FUNCTION_BLOCK "SINA_POS"   // FB1822, SCL
{ S7_Optimized_Access := 'TRUE' }
AUTHOR : DRVDPS7
FAMILY : DRIVES
NAME : SINA_POS
VERSION : 5.1
// stored: AutoNumber false, MemoryReserve 100, SetENOAutomatically false
   VAR_INPUT
      ModePos : Int := 0;   // 运行模式 1-相对；2-绝对；
      EnableAxis : Bool := 0;   // 使能驱动器
      CancelTraversing : Bool := 1;   // 0-取消当前任务运行;1-正常运行
      IntermediateStop : Bool := 1;   // 0-暂停当前的任务运行；1-正常运行
      Positive : Bool := 0;   // 正方向
      Negative : Bool := 0;   // 负方向
      Jog1 : Bool := 0;
      Jog2 : Bool := 0;
      FlyRef : Bool := 0;   // 激活被动寻零(CMMT不支持)
      AckError : Bool := 0;   // 故障复位
      ExecuteMode : Bool := 0;   // 激活ModPos模式
      Position : DInt := 0;   // 位置设定值或位置表行号
      Velocity : DInt := 0;   // 速度值
      OverV : Int := 100;   // 所有运动模式下的速度倍率（cmmt不支持）
      OverAcc : Int := 100;   // ModPos=1；2；3加速度百分比0-100
      OverDec : Int := 100;   // ModPos=1；2；3减速度百分比0-100
      ConfigEPos : DWord := 16#0000_0003;   // B0-3 功能位定义
      HWIDSTW : HW_IO := 0;   // CMMT 设备视图111报文硬件标识符
      HWIDZSW : HW_IO := 0;   // CMMT 设备视图111报文硬件标识符
   END_VAR
   VAR_OUTPUT
      AxisEnabled : Bool := 0;   // 驱动已经使能
      AxisPosOk : Bool := 0;   // 目标位置已到达
      AxisRef : Bool := 0;   // 已设置零点
      AxisWarn : Bool := 0;   // 驱动器报警
      AxisError : Bool := 0;   // 驱动器故障
      Lockout : Bool := 0;   // 驱动处于禁止接通状态，检查 ConfigEPos 第 0 位及第 1 位是否置 1
      ActVelocity : DInt := 0;   // 实际速度
      ActPosition : DInt := 0;   // 实际位置
      ActMode : Int := 0;   // 当前激活的模式
      EPosZSW1 : Word := 0;
      EPosZSW2 : Word := 0;
      ActWarn : Word := 0;   // 报警代码
      ActFault : Word := 0;   // 故障代码
      Error : Bool := 0;   // 功能块报错
      Status : Word := 0;   // 状态
      DiagID : Word := 0;   // 通信错误
   END_VAR
   VAR
      sbOff1Edge : Bool := 0;
      sbOff1 : Bool := 0;
      sbExecuteEdge : Bool := 0;
      sbExecute : Bool := 0;
      sbRefTypEdge : Bool := 0;
      sbRefTyp : Bool := 0;
      sbMdiStart : Bool := 0;
      sbMdiStartEdge : Bool := 0;
      sbRefStart : Bool := 0;
      sbJogInc : Bool := 0;
      sbReady : Bool := 0;
      sbIOp : Bool := 0;
      sbAccel : Bool := 0;
      sbDecel : Bool := 0;
      sbAlarm : Bool := 0;
      sbFault : Bool := 0;
      sbFWD : Bool := 0;
      sbBWD : Bool := 0;
      sbBusy : Bool := 0;
      swStatus : Word := 16#0000;
      swEPosZSW1 : Word := 16#0000;
      swEPosZSW2 : Word := 16#0000;
      siExecuteCyc : Int := 0;
      siRefTypCyc : Int := 0;
      siJogIncCyc : Int := 0;
      siMdiStartCyc : Int := 0;
      siRefActRetry : Int := 0;
      siModePos : Int := 0;
      siModePosMax : Int := 14;
      siCycWait : Int := 5;
      siRetryMax : Int := 15;
      sbModePos : Bool := 0;
      sxSendBuf : Struct
         STW1 : Word := WORD#16#0000;
         EPosSTW1 : Word := WORD#16#0000;
         EPosSTW2 : Word := WORD#16#0000;
         STW2 : Word := WORD#16#0000;
         OverrideV : Word := WORD#16#0000;
         Position : DWord := DWORD#16#0000_0000;
         Velocity : DWord := DWORD#16#0000_0000;
         OverrideA : Word := WORD#16#0000;
         OverrideD : Word := WORD#16#0000;
         Reserve : Word := WORD#16#0000;
      END_STRUCT;
      sxRecvBuf : Struct
         ZSW1 : Word := WORD#16#0000;
         EPosZSW1 : Word := WORD#16#0000;
         EPosZSW2 : Word := WORD#16#0000;
         ZSW2 : Word := WORD#16#0000;
         NotUsed : Word := WORD#16#0000;
         Position : DWord := DWORD#16#0000_0000;
         Velocity : DWord := DWORD#16#0000_0000;
         ErrNr : Word := WORD#16#0000;
         WarnNr : Word := WORD#16#0000;
         Reserve : Word := WORD#16#0000;
      END_STRUCT;
   END_VAR
   VAR_TEMP
      piRetSFC : Int;
      piCount : Int;
      swSendBuf : Array[0..11] of Word;
      swRecvBuf : Array[0..11] of Word;
   END_VAR
BEGIN

   //=============================================================================
   //SIEMENS AG
   //(c)Copyright 2017 All Rights Reserved
   //-----------------------------------------------------------------------------
   // Library: DriveLib
   // Tested with: S7-1516-3 PN/DP V1.8
   // Engineering: TIA Portal V14
   // Restrictions: -
   // Requirements: S7-1200 / S7-1500
   // Functionality: cyclic communication between a SINAMICS (Basic positioner)and a PLC
   //                If in HWConfig Std.TLG 111 is projected 12 PZD-words are exchanged
   //                in every bus cycle.
   //                The parametrisation of these words is described in the manual of the
   //                SINAMICS
   //=============================================================================

   // Betriebsart ermitteln
   IF #ModePos > #siModePosMax THEN

     #sbModePos := FALSE;
     #Error := True;
     #swStatus := 16#8202;//不正确的运行模式
   ELSIF #ModePos < 1 THEN

     #sbModePos := FALSE;
     #Error := True;
     #swStatus := 16#8202;//不正确的运行模式
   ELSE
     // Betriebsartenwechsel ist nur möglich, wenn die Achse nicht beschleunigt oder nicht verzögert 
     // und die Geschwindigkeit Null ist
     IF NOT #sbFWD AND NOT #sbBWD AND NOT #sbAccel AND NOT #sbDecel THEN

       #sbModePos := TRUE;
       #siModePos := #ModePos;

       // Fehler wieder zurücknehmen, wenn er mal ausgelöst wurde
       IF #swStatus = 16#8202 THEN
           #swStatus := 16#7002;//功能块正常执行
         #Error := False;
       END_IF;
     END_IF;
   END_IF;

   // Überprüfung der analogen Eingabewerte, ob sie innerhalb des möglichen Bereiches liegen
   // Geschwindigkeitsoverride (0% - 199%, 100% => W#16#4000)
   IF (#OverV < 0) OR (#OverV > 199) THEN
       #swStatus := 16#8203;//参数设置错误
     #Error := True;
   ELSE
     // Geschwindigkeitsoverride in den Sendepuffer eintragen
     #sxSendBuf.OverrideV := INT_TO_WORD(REAL_TO_INT(16384.0 * (INT_TO_REAL(#OverV) / 100.0)));
   END_IF;

   // Beschleunigungsoverride (0% - 100%, 100% => W#16#4000)
   IF (#OverAcc < 0) OR (#OverAcc > 100) THEN
       #swStatus := 16#8203;//参数设置错误
     #Error := True;
   ELSE
     // Beschleunigungsoverride in den Sendepuffer eintragen
     #sxSendBuf.OverrideA := INT_TO_WORD(REAL_TO_INT(16384.0 * (INT_TO_REAL(#OverAcc) / 100.0)));
   END_IF;

   // Verzögerungsoverride (0% - 100%, 100% => W#16#4000)
   IF (#OverDec < 0) OR (#OverDec > 100) THEN
       #swStatus := 16#8203;//参数设置错误
     #Error := True;
   ELSE
     // Verzögerungsoverride in den Sendepuffer eintragen
     #sxSendBuf.OverrideD := INT_TO_WORD(REAL_TO_INT(16384.0 * (INT_TO_REAL(#OverDec) / 100.0)));
   END_IF;

   // Fehler wieder zurücknehmen, wenn er mal ausgelöst wurde
   IF NOT (#OverV < 0) AND NOT (#OverV > 199) AND NOT (#OverAcc < 0) AND NOT (#OverAcc > 100) AND
     NOT (#OverDec < 0) AND NOT (#OverDec > 100) THEN
     IF #swStatus = 16#8203 THEN
       #swStatus := 16#7002;
       #Error := False;
     END_IF;
   END_IF;

   // Positionssollwert
   // Positionssollwert in den Sendepuffer eintragen
   #sxSendBuf.Position := DINT_TO_DWORD(#Position);

   // Geschwindigkeitssollwert (Begrenzung / Überwachung
   // Geschwindigkeitssollwert in den Sendepuffer eintragen
   #sxSendBuf.Velocity := DINT_TO_DWORD(#Velocity);

   // Einschalten bzw. Ausschalten des Antriebes erkennen
   IF #EnableAxis AND NOT #sbOff1Edge AND NOT #sbBusy AND #sbModePos THEN
     #sbOff1 := True;
   END_IF;
   // Einschalten bzw. Ausschalten des Antriebes Flanke merken
   #sbOff1Edge := #EnableAxis AND NOT #sbBusy;

   // Einschaltflankenmerker wieder zurücksetzen
   IF NOT #EnableAxis THEN
     #sbOff1 := False;
   END_IF;

   // Fliegendes Referenzieren aktivieren erkennen
   IF #FlyRef AND NOT #sbRefTypEdge THEN
     #sbRefTyp := True;
   END_IF;
   // Fliegendes Referenzieren aktivieren Flanke merken
   #sbRefTypEdge := #FlyRef;

   // Fliegendes Referenzieren Flankenmerker wieder zurücksetzen
   IF NOT #FlyRef THEN
     #sbRefTyp := False;
     #siRefTypCyc := 0;
   END_IF;

   // Verfahrauftrag aktivieren erkennen
   IF #ExecuteMode AND NOT #sbExecuteEdge THEN
     #sbExecute := True;
   END_IF;
   // Verfahrauftrag aktivieren Flanke merken
   #sbExecuteEdge := #ExecuteMode;

   // Verfahrauftragflankenmerker wieder zurücksetzen
   IF NOT #ExecuteMode THEN
     #sbExecute := False;
     #siExecuteCyc := 0;
   END_IF;

   // Betriebsart MDI / Sollwertdirektvorgabe Flanke merken
   (*IF #sxSendBuf.sxEPosSTW1.MdiStart AND NOT #sbMdiStartEdge THEN
             #sbMdiStart := True;
         END_IF;
         // Betriebsart MDI / Sollwertdirektvorgabe Flanke merken
         #sbMdiStartEdge := #sxSendBuf.sxEPosSTW1.MdiStart AND NOT #Busy;*)

   // Verfahrauftragflankenmerker wieder zurücksetzen
   (*IF NOT #sxSendBuf.sxEPosSTW1.MdiStart THEN
             #sbMdiStart := False;
             #siMdiStartCyc := 0;
         END_IF;*)

   IF #sxSendBuf.EPosSTW1.%X15 AND NOT #sbMdiStartEdge THEN
     #sbMdiStart := True;
   END_IF;
   // Betriebsart MDI / Sollwertdirektvorgabe Flanke merken
   #sbMdiStartEdge := #sxSendBuf.EPosSTW1.%X15 AND NOT #sbBusy;

   // Verfahrauftragflankenmerker wieder zurücksetzen
   IF NOT #sxSendBuf.EPosSTW1.%X15 THEN
     #sbMdiStart := False;
     #siMdiStartCyc := 0;
   END_IF;

   // Schreibdaten zusammenstellen
   // Steuerword STW1 für alle Betriebsart aufbereiten
   (*#sxSendBuf.sxSTW1.RejTrvTsk        := #RejTrvTsk;
         #sxSendBuf.sxSTW1.IntMStop         := #IntMStop;
         #sxSendBuf.sxSTW1.AckFault         := #AckFlt;*)

   #sxSendBuf.STW1.%X4 := #CancelTraversing;
   #sxSendBuf.STW1.%X5 := #IntermediateStop;
   #sxSendBuf.STW1.%X7 := #AckError;
   #sxSendBuf.STW1.%X1 := TRUE;
   #sxSendBuf.STW1.%X2 := TRUE;
   #sxSendBuf.STW1.%X3 := TRUE;
   #sxSendBuf.STW1.%X10 := TRUE;

   // Hauptbetriebsart "Positionieren / manueller Sollwertvorgabe (MDI)" 
   // Betriebsart "Positionieren Relativ positiv" oder "Positionieren Relativ negativ"
   IF (#siModePos = 1 AND #sbModePos) THEN

     // Antrieb einschalten
     //#sxSendBuf.sxSTW1.Off1 := #sbOff1;
     #sxSendBuf.STW1.%X0 := #sbOff1;

     // nicht verwendete Signale für den 1. Schritt und eventuell weitere Schritte
     (*#sxSendBuf.sxSTW1.Jog1          := False;
             #sxSendBuf.sxSTW1.Jog2          := False;
             #sxSendBuf.sxEPosSTW1.MdiTyp    := False;
             #sxSendBuf.sxEPosSTW1.MdiPos    := False;
             #sxSendBuf.sxEPosSTW1.MdiNeg    := False;
             #sxSendBuf.sxEPosSTW1.MdiSetup  := False;
             #sxSendBuf.sxEPosSTW2.SetRefPt  := False;
             #sxSendBuf.sxEPosSTW2.JogInc    := False;
             #sxSendBuf.sxEPosSTW2.RefStDi   := False;
             #sxSendBuf.sxSTW1.RefStart      := False;
             #sxSendBuf.sxEPosSTW2.RefTyp    := False;
             #sxSendBuf.sxEPosSTW1.MdiStart  := False;*)
     #sxSendBuf.STW1.%X8 := False;
     #sxSendBuf.STW1.%X9 := False;
     #sxSendBuf.EPosSTW1.%X8 := False;
     #sxSendBuf.EPosSTW1.%X9 := False;
     #sxSendBuf.EPosSTW1.%X10 := False;
     #sxSendBuf.EPosSTW1.%X14 := False;
     #sxSendBuf.EPosSTW2.%X1 := False;
     #sxSendBuf.EPosSTW2.%X5 := False;
     #sxSendBuf.EPosSTW2.%X9 := False;
     #sxSendBuf.STW1.%X11 := False;
     #sxSendBuf.EPosSTW2.%X8 := False;
     #sxSendBuf.EPosSTW1.%X15 := False;


     // Nach dem Einschalten des Antriebes, prüfen ob der Antrieb betriebsbereit, in Operation ohne Fehler und Warnung ist, 
     // dann die Betriebsart MDI / Sollwertvorgabe Start gesetzt werden
     IF #sbOff1 AND #sbReady AND #sbIOp AND NOT #sbFault THEN

       // Betriebsart MDI / Sollwertdirektvorgabe setzen
       //#sxSendBuf.sxEPosSTW1.MdiStart := True;
       #sxSendBuf.EPosSTW1.%X15 := True;

       // Positioniertyp auf relatives Positionieren stellen 
       //#sxSendBuf.sxEPosSTW1.MdiTyp := False;
       #sxSendBuf.EPosSTW1.%X8 := False;

       // die Richtungswahl für das Positionieren auf positive Richtung oder negative Richtung einstellen
       IF #Positive AND NOT #Negative THEN

         // positive Richtung
         //#sxSendBuf.sxEPosSTW1.MdiPos := True;
         #sxSendBuf.EPosSTW1.%X9 := True;

         // negative Richtung
         //#sxSendBuf.sxEPosSTW1.MdiNeg := False;
         #sxSendBuf.EPosSTW1.%X10 := False;

         // die Richtungswahl für das Positionieren auf negative Richtung einstellen                
       ELSIF NOT #Positive AND #Negative THEN

         // positive Richtung
         //#sxSendBuf.sxEPosSTW1.MdiPos := False;
         #sxSendBuf.EPosSTW1.%X9 := False;

         // negative Richtung
         //#sxSendBuf.sxEPosSTW1.MdiNeg := True;
         #sxSendBuf.EPosSTW1.%X10 := True;

         // die Richtungswahl für das Positionieren auf keine Richtung einstellen                
       ELSE

         // positive Richtung
         //#sxSendBuf.sxEPosSTW1.MdiPos := False;
         #sxSendBuf.EPosSTW1.%X9 := False;

         // negative Richtung
         //#sxSendBuf.sxEPosSTW1.MdiNeg := False;
         #sxSendBuf.EPosSTW1.%X10 := False;

       END_IF;

       // Nach dem Einschalten des Antriebes und dem Betriebsart MDI / Sollwertvorgabe starten, 
       // ein Paar Zyklen warten bevor die Flanke für die Sollwertübernahme MDI gesetzt werden kann
       IF #sbMdiStart AND (#siMdiStartCyc < #siCycWait) THEN
         #siMdiStartCyc := #siMdiStartCyc + 1;
       ELSE
         // Flanke Sollwertübernahme MDI
         //#sxSendBuf.sxSTW1.TrvStart := #Execute;
         #sxSendBuf.STW1.%X6 := #ExecuteMode;

       END_IF;

       // "Fliegendes Referentieren" aktivieren
       // "Fliegendes Referenzieren" erst nach Einschalten des Antriebes möglich
       IF #sbRefTyp THEN

         // Referenziertyp auf "Fliegendes Referenzieren" einstellen
         //#sxSendBuf.sxEPosSTW2.RefTyp := True;
         #sxSendBuf.EPosSTW2.%X8 := True;

         // Nach der Anwahl des Referenziertyps "Fliegendes Referenzieren", 
         // ein Zyklus später kann das Referenzieren gestartet
         IF (#siRefTypCyc = 0) THEN
           #siRefTypCyc := #siRefTypCyc + 1;
         ELSE
           // Referenzieren starten
           //#sxSendBuf.sxSTW1.RefStart := True;
           #sxSendBuf.STW1.%X11 := True;

         END_IF;
       END_IF;
     END_IF;

     // Betriebsart "Positionieren Absolut" oder "Positonieren Absolut positiv" oder "Positionieren Absolut negativ"
   ELSIF #siModePos = 2 AND #sbModePos THEN

     // Antrieb einschalten
     //#sxSendBuf.sxSTW1.Off1 := #sbOff1;
     #sxSendBuf.STW1.%X0 := #sbOff1;

     // nicht verwendete Signale für den 1. Schritt und eventuell weitere Schritte
     (*#sxSendBuf.sxSTW1.Jog1         := False;
             #sxSendBuf.sxSTW1.Jog2         := False;
             #sxSendBuf.sxEPosSTW1.MdiTyp   := False;
             #sxSendBuf.sxEPosSTW1.MdiPos   := False;
             #sxSendBuf.sxEPosSTW1.MdiNeg   := False;
             #sxSendBuf.sxEPosSTW1.MdiSetup := False;
             #sxSendBuf.sxEPosSTW2.SetRefPt := False;
             #sxSendBuf.sxEPosSTW2.JogInc   := False;
             #sxSendBuf.sxEPosSTW2.RefStDi  := False;
             #sxSendBuf.sxSTW1.RefStart     := False;
             #sxSendBuf.sxEPosSTW2.RefTyp   := False;
             #sxSendBuf.sxEPosSTW1.MdiStart := False;*)
     #sxSendBuf.STW1.%X8 := False;
     #sxSendBuf.STW1.%X9 := False;
     #sxSendBuf.EPosSTW1.%X8 := False;
     #sxSendBuf.EPosSTW1.%X9 := False;
     #sxSendBuf.EPosSTW1.%X10 := False;
     #sxSendBuf.EPosSTW1.%X14 := False;
     #sxSendBuf.EPosSTW2.%X1 := False;
     #sxSendBuf.EPosSTW2.%X5 := False;
     #sxSendBuf.EPosSTW2.%X9 := False;
     #sxSendBuf.STW1.%X11 := False;
     #sxSendBuf.EPosSTW2.%X8 := False;
     #sxSendBuf.EPosSTW1.%X15 := False;

     // Nach dem Einschalten des Antriebes, prüfen ob der Antrieb betriebsbereit, in Operation ohne Fehler und Warnung ist, 
     // dann die Betriebsart MDI / Sollwertvorgabe Start gesetzt werden
     IF #sbOff1 AND #sbReady AND #sbIOp AND NOT #sbFault THEN

       // Betriebsart MDI / Sollwertdirektvorgabe setzen
       //#sxSendBuf.sxEPosSTW1.MdiStart := True;
       #sxSendBuf.EPosSTW1.%X15 := True;

       // Positioniertyp auf absolutes Positionieren stellen 
       //#sxSendBuf.sxEPosSTW1.MdiTyp := True;
       #sxSendBuf.EPosSTW1.%X8 := True;

       // die Richtungswahl für das Positionieren auf positive Richtung oder negative Richtung einstellen
       IF #Positive AND NOT #Negative THEN

         // positive Richtung
         //#sxSendBuf.sxEPosSTW1.MdiPos := True;
         #sxSendBuf.EPosSTW1.%X9 := True;

         // negative Richtung
         //#sxSendBuf.sxEPosSTW1.MdiNeg := False;
         #sxSendBuf.EPosSTW1.%X10 := False;

         // die Richtungswahl für das Positionieren auf negative Richtung einstellen                
       ELSIF NOT #Positive AND #Negative THEN

         // positive Richtung
         //#sxSendBuf.sxEPosSTW1.MdiPos := False;
         #sxSendBuf.EPosSTW1.%X9 := False;

         // negative Richtung
         //#sxSendBuf.sxEPosSTW1.MdiNeg := True;
         #sxSendBuf.EPosSTW1.%X10 := True;

         // die Richtungswahl für das Positionieren auf keine Richtung einstellen                
       ELSE

         // positive Richtung
         //#sxSendBuf.sxEPosSTW1.MdiPos := False;
         #sxSendBuf.EPosSTW1.%X9 := False;

         // negative Richtung
         //#sxSendBuf.sxEPosSTW1.MdiNeg := False;
         #sxSendBuf.EPosSTW1.%X10 := False;

       END_IF;

       // Nach dem Einschalten des Antriebes und dem Betriebsart MDI / Sollwertvorgabe starten, 
       // ein Paar Zyklen warten bevor die Flanke für die Sollwertübernahme MDI gesetzt werden kann
       IF #sbMdiStart AND (#siMdiStartCyc < #siCycWait) THEN
         #siMdiStartCyc := #siMdiStartCyc + 1;
       ELSE
         // Flanke Sollwertübernahme MDI
         //#sxSendBuf.sxSTW1.TrvStart := #Execute;
         #sxSendBuf.STW1.%X6 := #ExecuteMode;

       END_IF;

       // "Fliegendes Referentieren" aktivieren
       // "Fliegendes Referenzieren" erst nach Einschalten des Antriebes möglich
       IF #sbRefTyp THEN

         // Referenziertyp auf "Fliegendes Referenzieren" einstellen
         //#sxSendBuf.sxEPosSTW2.RefTyp := True;
         #sxSendBuf.EPosSTW2.%X8 := True;

         // Nach der Anwahl des Referenziertyps "Fliegendes Referenzieren", 
         // ein Zyklus später kann das Referenzieren gestartet
         IF (#siRefTypCyc = 0) THEN
           #siRefTypCyc := #siRefTypCyc + 1;
         ELSE
           // Referenzieren starten
           //#sxSendBuf.sxSTW1.RefStart := True;
           #sxSendBuf.STW1.%X11 := True;

         END_IF;
       END_IF;
     END_IF;

     // Betriebsart "Positionieren als Einrichten positiv" oder "Positionieren als Einrichten negativ"
   ELSIF #siModePos = 3 AND #sbModePos THEN

     // Antrieb einschalten
     //#sxSendBuf.sxSTW1.Off1 := #sbOff1;
     #sxSendBuf.STW1.%X0 := #sbOff1;

     // nicht verwendete Signale für den 1. Schritt und eventuell weitere Schritte
     (*#sxSendBuf.sxSTW1.Jog1           := False;
             #sxSendBuf.sxSTW1.Jog2           := False;
             #sxSendBuf.sxEPosSTW1.MdiTyp     := False;
             #sxSendBuf.sxEPosSTW1.MdiPos     := False;
             #sxSendBuf.sxEPosSTW1.MdiNeg     := False;
             #sxSendBuf.sxEPosSTW1.MdiSetup   := False;
             #sxSendBuf.sxEPosSTW2.SetRefPt   := False;
             #sxSendBuf.sxEPosSTW2.JogInc     := False;
             #sxSendBuf.sxEPosSTW2.RefStDi    := False;
             #sxSendBuf.sxSTW1.RefStart       := False;
             #sxSendBuf.sxEPosSTW2.RefTyp     := False;
             #sxSendBuf.sxEPosSTW1.MdiStart   := False;*)
     #sxSendBuf.STW1.%X8 := False;
     #sxSendBuf.STW1.%X9 := False;
     #sxSendBuf.EPosSTW1.%X8 := False;
     #sxSendBuf.EPosSTW1.%X9 := False;
     #sxSendBuf.EPosSTW1.%X10 := False;
     #sxSendBuf.EPosSTW1.%X14 := False;
     #sxSendBuf.EPosSTW2.%X1 := False;
     #sxSendBuf.EPosSTW2.%X5 := False;
     #sxSendBuf.EPosSTW2.%X9 := False;
     #sxSendBuf.STW1.%X11 := False;
     #sxSendBuf.EPosSTW2.%X8 := False;
     #sxSendBuf.EPosSTW1.%X15 := False;

     // Nach dem Einschalten des Antriebes, prüfen ob der Antrieb betriebsbereit, in Operation ohne Fehler und Warnung ist, 
     // dann die Betriebsart MDI / Sollwertvorgabe Start gesetzt werden
     IF #sbOff1 AND #sbReady AND #sbIOp AND NOT #sbFault THEN

       // Betriebsart MDI / Sollwertdirektvorgabe setzen
       //#sxSendBuf.sxEPosSTW1.MdiStart := True;
       #sxSendBuf.EPosSTW1.%X15 := True;

       // Positioniertyp auf absolutes Positionieren stellen 
       //#sxSendBuf.sxEPosSTW1.MdiTyp := True;
       #sxSendBuf.EPosSTW1.%X8 := True;

       // die Anwahl für MDI Modus auf Einrichten einstellen
       //#sxSendBuf.sxEPosSTW1.MdiSetup := True;
       #sxSendBuf.EPosSTW1.%X14 := True;

       // die Richtungswahl für das Positionieren auf positive Richtung oder negative Richtung einstellen
       IF #Positive AND NOT #Negative THEN

         // positive Richtung
         //#sxSendBuf.sxEPosSTW1.MdiPos := True;
         #sxSendBuf.EPosSTW1.%X9 := True;

         // negative Richtung
         //#sxSendBuf.sxEPosSTW1.MdiNeg := False;
         #sxSendBuf.EPosSTW1.%X10 := False;

         // die Richtungswahl für das Positionieren auf negative Richtung einstellen                
       ELSIF NOT #Positive AND #Negative THEN

         // positive Richtung
         //#sxSendBuf.sxEPosSTW1.MdiPos := False;
         #sxSendBuf.EPosSTW1.%X9 := False;

         // negative Richtung
         //#sxSendBuf.sxEPosSTW1.MdiNeg := True;
         #sxSendBuf.EPosSTW1.%X10 := True;

         // die Richtungswahl für das Positionieren auf keine Richtung einstellen                
       ELSE

         // positive Richtung
         //#sxSendBuf.sxEPosSTW1.MdiPos := False;
         #sxSendBuf.EPosSTW1.%X9 := False;

         // negative Richtung
         //#sxSendBuf.sxEPosSTW1.MdiNeg := False;
         #sxSendBuf.EPosSTW1.%X10 := False;

       END_IF;

       // Nach dem Einschalten des Antriebes und dem Betriebsart MDI / Sollwertvorgabe starten, 
       // ein Paar Zyklen warten bevor die Flanke für die Sollwertübernahme MDI gesetzt werden kann
       IF #sbMdiStart AND (#siMdiStartCyc < #siCycWait) THEN
         #siMdiStartCyc := #siMdiStartCyc + 1;
       ELSE
         // Flanke Sollwertübernahme MDI
         //#sxSendBuf.sxSTW1.TrvStart := #Execute;
         #sxSendBuf.STW1.%X6 := #ExecuteMode;

       END_IF;

       // "Fliegendes Referentieren" aktivieren
       // "Fliegendes Referenzieren" erst nach Einschalten des Antriebes möglich
       IF #sbRefTyp THEN

         // Referenziertyp auf "Fliegendes Referenzieren" einstellen
         //#sxSendBuf.sxEPosSTW2.RefTyp := True;
         #sxSendBuf.EPosSTW2.%X8 := True;

         // Nach der Anwahl des Referenziertyps "Fliegendes Referenzieren", 
         // ein Zyklus später kann das Referenzieren gestartet
         IF (#siRefTypCyc = 0) THEN
           #siRefTypCyc := #siRefTypCyc + 1;
         ELSE
           // Referenzieren starten
           //#sxSendBuf.sxSTW1.RefStart := True;
           #sxSendBuf.STW1.%X11 := True;

         END_IF;
       END_IF;
     END_IF;

     // Hauptbetriebsart "Referenzieren" (Reference)
     // Betriebsart "Referenzieren - Referenzpunktfahrt positiv" oder "Referenzieren - Referenzpunktfahrt negativ"
   ELSIF #siModePos = 4 AND #sbModePos THEN

     // Antrieb einschalten
     //#sxSendBuf.sxSTW1.Off1 := #sbOff1;
     #sxSendBuf.STW1.%X0 := #sbOff1;

     // nicht verwendete Signale für den 1. Schritt und eventuell weitere Schritte
     (*#sxSendBuf.sxSTW1.Jog1         := False;
             #sxSendBuf.sxSTW1.Jog2         := False;
             #sxSendBuf.sxEPosSTW1.MdiStart := False;
             #sxSendBuf.sxEPosSTW2.SetRefPt := False;
             #sxSendBuf.sxEPosSTW2.JogInc   := False;
             #sxSendBuf.sxEPosSTW2.RefTyp   := False;
             #sxSendBuf.sxSTW1.RefStart     := False;
             #sxSendBuf.sxEPosSTW2.RefStDi  := False;*)
     #sxSendBuf.STW1.%X8 := False;
     #sxSendBuf.STW1.%X9 := False;
     #sxSendBuf.EPosSTW1.%X15 := False;
     #sxSendBuf.EPosSTW2.%X1 := False;
     #sxSendBuf.EPosSTW2.%X5 := False;
     #sxSendBuf.EPosSTW2.%X8 := False;
     #sxSendBuf.STW1.%X11 := False;
     #sxSendBuf.EPosSTW2.%X9 := False;

     // Nach dem Einschalten des Antriebes, prüfen ob der Antrieb betriebsbereit, in Operation ohne Fehler und Warnung ist, 
     // dann die Betriebsart MDI / Sollwertvorgabe Start gesetzt werden
     IF #sbOff1 AND #sbReady AND #sbIOp AND NOT #sbFault THEN

       // Referenzieren starten
       //#sxSendBuf.sxSTW1.RefStart := #Execute;
       #sxSendBuf.STW1.%X11 := #ExecuteMode;

       // die Richtungswahl für das Referenzpunktfahrt positiv einstellen
       IF #Positive AND NOT #Negative THEN

         // positive Referenzpunktfahrt
         //#sxSendBuf.sxEPosSTW2.RefStDi := False;
         #sxSendBuf.EPosSTW2.%X9 := False;

         // die Richtungswahl für das Referenzpunktfahrt negativ einstellen                
       ELSIF NOT #Positive AND #Negative THEN

         // negative Referenzpunktfahrt
         //#sxSendBuf.sxEPosSTW2.RefStDi := True;
         #sxSendBuf.EPosSTW2.%X9 := True;

       END_IF;
     END_IF;

     // Betriebsart "Referenzieren - Referenzpunkt setzen"
   ELSIF #siModePos = 5 AND #sbModePos THEN

     // Antrieb einschalten
     //#sxSendBuf.sxSTW1.Off1 := #sbOff1;
     #sxSendBuf.STW1.%X0 := #sbOff1;

     // nicht verwendete Signale für den 1. Schritt und eventuell weitere Schritte
     (*#sxSendBuf.sxSTW1.Jog1          := False;
             #sxSendBuf.sxSTW1.Jog2          := False;
             #sxSendBuf.sxSTW1.RefStart      := False;
             #sxSendBuf.sxEPosSTW1.MdiStart  := False;
             #sxSendBuf.sxEPosSTW2.JogInc    := False;
             #sxSendBuf.sxEPosSTW2.RefTyp    := False;
             #sxSendBuf.sxEPosSTW2.RefStDi   := False;
             #sxSendBuf.sxEPosSTW2.SetRefPt  := False;*)
     #sxSendBuf.STW1.%X8 := False;
     #sxSendBuf.STW1.%X9 := False;
     #sxSendBuf.STW1.%X11 := False;
     #sxSendBuf.EPosSTW1.%X15 := False;
     #sxSendBuf.EPosSTW2.%X5 := False;
     #sxSendBuf.EPosSTW2.%X8 := False;
     #sxSendBuf.EPosSTW2.%X9 := False;
     #sxSendBuf.EPosSTW2.%X1 := False;

     // Nach dem Einschalten des Antriebes, prüfen ob der Antrieb betriebsbereit, in Operation ohne Fehler und Warnung ist, 
     // dann die Betriebsart MDI / Sollwertvorgabe Start gesetzt werden
     IF NOT #sbFault THEN

       // Referenzpunktfahrt negativ
       //#sxSendBuf.sxEPosSTW2.SetRefPt := #Execute;
       #sxSendBuf.EPosSTW2.%X1 := #ExecuteMode;

     END_IF;

     // Hauptbetriebsart "Verfahrsätze" (Traversing Blocks)
   ELSIF #siModePos = 6 AND #sbModePos THEN

     // Antrieb einschalten
     //#sxSendBuf.sxSTW1.Off1 := #sbOff1;
     #sxSendBuf.STW1.%X0 := #sbOff1;

     // nicht verwendete Signale für den 1. Schritt und eventuell weitere Schritte
     (*#sxSendBuf.sxSTW1.Jog1          := False;
             #sxSendBuf.sxSTW1.Jog2          := False;
             #sxSendBuf.sxEPosSTW1.MdiTyp    := False;
             #sxSendBuf.sxEPosSTW1.MdiPos    := False;
             #sxSendBuf.sxEPosSTW1.MdiNeg    := False;
             #sxSendBuf.sxEPosSTW1.MdiSetup  := False;
             #sxSendBuf.sxEPosSTW2.SetRefPt  := False;
             #sxSendBuf.sxEPosSTW2.JogInc    := False;
             #sxSendBuf.sxEPosSTW2.RefStDi   := False;
             #sxSendBuf.sxEPosSTW2.RefTyp    := False;
             #sxSendBuf.sxSTW1.RefStart      := False;
             #sxSendBuf.sxEPosSTW1.TrvBit0   := False;
             #sxSendBuf.sxEPosSTW1.TrvBit1   := False;
             #sxSendBuf.sxEPosSTW1.TrvBit2   := False;
             #sxSendBuf.sxEPosSTW1.TrvBit3   := False;
             #sxSendBuf.sxEPosSTW1.TrvBit4   := False;
             #sxSendBuf.sxEPosSTW1.TrvBit5   := False;
             #sxSendBuf.sxEPosSTW1.MdiStart  := False;*)
     #sxSendBuf.STW1.%X8 := False;
     #sxSendBuf.STW1.%X9 := False;
     #sxSendBuf.EPosSTW1.%X8 := False;
     #sxSendBuf.EPosSTW1.%X9 := False;
     #sxSendBuf.EPosSTW1.%X10 := False;
     #sxSendBuf.EPosSTW1.%X14 := False;
     #sxSendBuf.EPosSTW2.%X1 := False;
     #sxSendBuf.EPosSTW2.%X5 := False;
     #sxSendBuf.EPosSTW2.%X9 := False;
     #sxSendBuf.EPosSTW2.%X8 := False;
     #sxSendBuf.STW1.%X11 := False;
     #sxSendBuf.EPosSTW1.%X0 := False;
     #sxSendBuf.EPosSTW1.%X1 := False;
     #sxSendBuf.EPosSTW1.%X2 := False;
     #sxSendBuf.EPosSTW1.%X3 := False;
     #sxSendBuf.EPosSTW1.%X4 := False;
     #sxSendBuf.EPosSTW1.%X5 := False;
     #sxSendBuf.EPosSTW1.%X15 := False;

     // Bei der Auswahl der Verfahrsätze entspricht die Position der Verfahrensatznummer 
     // Verfahrsatznummer aus der Position ermitteln und in die einzelnen Bit's aufteilen
     // Es sind die Verfahrsatznummern 0 - 63 möglich
     IF (DINT_TO_INT(#Position) < 0) OR (DINT_TO_INT(#Position) > 63) THEN
       // Fehler, ungültiger Verfahrsatznummer
       #swStatus := 16#8204;
       #Error := True;
     ELSE
       // Fehler wieder zurücknehmen, wenn er mal ausgelöst wurde
       IF #swStatus = 16#8204 THEN
         #swStatus := 16#7002;
         #Error := False;
       END_IF;

       // Verfahrsatznummer Bit 0 ermitteln
       IF (DINT_TO_WORD(#Position) AND W#16#01) = W#16#01 THEN
         //#sxSendBuf.sxEPosSTW1.TrvBit0 := True;
         #sxSendBuf.EPosSTW1.%X0 := True;
       END_IF;

       // Verfahrsatznummer Bit 1 ermitteln
       IF (DINT_TO_WORD(#Position) AND W#16#02) = W#16#02 THEN
         //#sxSendBuf.sxEPosSTW1.TrvBit1 := True;
         #sxSendBuf.EPosSTW1.%X1 := True;
       END_IF;

       // Verfahrsatznummer Bit 2 ermitteln
       IF (DINT_TO_WORD(#Position) AND W#16#04) = W#16#04 THEN
         //#sxSendBuf.sxEPosSTW1.TrvBit2 := True;
         #sxSendBuf.EPosSTW1.%X2 := True;
       END_IF;

       // Verfahrsatznummer Bit 3 ermitteln
       IF (DINT_TO_WORD(#Position) AND W#16#08) = W#16#08 THEN
         //#sxSendBuf.sxEPosSTW1.TrvBit3 := True;
         #sxSendBuf.EPosSTW1.%X3 := True;
       END_IF;

       // Verfahrsatznummer Bit 4 ermitteln
       IF (DINT_TO_WORD(#Position) AND W#16#10) = W#16#10 THEN
         //#sxSendBuf.sxEPosSTW1.TrvBit4 := True;
         #sxSendBuf.EPosSTW1.%X4 := True;
       END_IF;

       // Verfahrsatznummer Bit 5 ermitteln
       IF (DINT_TO_WORD(#Position) AND W#16#20) = W#16#20 THEN
         //#sxSendBuf.sxEPosSTW1.TrvBit5 := True;
         #sxSendBuf.EPosSTW1.%X5 := True;
       END_IF;

       // Nach dem Einschalten des Antriebes, prüfen ob der Antrieb betriebsbereit, in Operation ohne Fehler und Warnung ist, 
       // dann die Betriebsart MDI / Sollwertvorgabe Start gesetzt werden
       IF #sbOff1 AND #sbReady AND #sbIOp AND NOT #sbFault THEN

         // Positioniertyp auf absolutes Positionieren stellen 
         //#sxSendBuf.sxEPosSTW1.MdiTyp := True;
         #sxSendBuf.EPosSTW1.%X8 := True;

         // die Richtungswahl für das Positionieren auf positive Richtung einstellen
         //#sxSendBuf.sxEPosSTW1.MdiPos := True;
         #sxSendBuf.EPosSTW1.%X9 := True;

         // die Richtungswahl für das Positionieren auf negative Richtung abstellen
         //#sxSendBuf.sxEPosSTW1.MdiNeg := False;
         #sxSendBuf.EPosSTW1.%X10 := False;

         // die Anwahl für MDI Modus auf Einrichten einstellen
         //#sxSendBuf.sxEPosSTW1.MdiSetup := True;
         #sxSendBuf.EPosSTW1.%X14 := True;

         // Nach dem Einschalten des Antriebes und dem Betriebsart MDI / Sollwertvorgabe starten, 
         // ein Paar Zyklen warten bevor die Flanke für die Sollwertübernahme MDI gesetzt werden kann
         IF #sbMdiStart AND (#siMdiStartCyc < #siCycWait) THEN
           #siMdiStartCyc := #siMdiStartCyc + 1;
         ELSE
           // Flanke Sollwertübernahme MDI
           //#sxSendBuf.sxSTW1.TrvStart := #Execute;
           #sxSendBuf.STW1.%X6 := #ExecuteMode;
         END_IF;

         // "Fliegendes Referentieren" aktivieren
         // "Fliegendes Referenzieren" erst nach Einschalten des Antriebes möglich
         IF #sbRefTyp THEN

           // Referenziertyp auf "Fliegendes Referenzieren" einstellen
           //#sxSendBuf.sxEPosSTW2.RefTyp := True;
           #sxSendBuf.EPosSTW2.%X8 := True;

           // Nach der Anwahl des Referenziertyps "Fliegendes Referenzieren", 
           // ein Zyklus später kann das Referenzieren gestartet
           IF (#siRefTypCyc = 0) THEN
             #siRefTypCyc := #siRefTypCyc + 1;
           ELSE
             // Referenzieren starten
             //#sxSendBuf.sxSTW1.RefStart := True;
             #sxSendBuf.STW1.%X11 := True;
           END_IF;
         END_IF;
       END_IF;
     END_IF;

     // Hauptbetriebsart "Tippen" (Jogging)
     // Betriebsart "Tippen positiv" oder "Tippen negativ" angewählt 
   ELSIF #siModePos = 7 AND #sbModePos THEN

     // Antrieb einschalten
     //#sxSendBuf.sxSTW1.Off1 := #sbOff1;
     #sxSendBuf.STW1.%X0 := #sbOff1;

     // nicht verwendete Signale für den 1. Schritt und eventuell weitere Schritte
     (*#sxSendBuf.sxEPosSTW1.MdiStart := False;
             #sxSendBuf.sxEPosSTW2.JogInc   := False;
             #sxSendBuf.sxSTW1.Jog1         := False;
             #sxSendBuf.sxSTW1.Jog2         := False;
             #sxSendBuf.sxEPosSTW2.RefTyp   := False;
             #sxSendBuf.sxSTW1.RefStart     := False;*)

     #sxSendBuf.EPosSTW1.%X15 := False;
     #sxSendBuf.EPosSTW2.%X5 := False;
     #sxSendBuf.STW1.%X8 := False;
     #sxSendBuf.STW1.%X9 := False;
     #sxSendBuf.EPosSTW2.%X8 := False;
     #sxSendBuf.STW1.%X11 := False;

     // Nach dem Einschalten des Antriebes, prüfen ob der Antrieb betriebsbereit, in Operation ohne Fehler und Warnung ist, 
     // dann kann Tippen positiv oder negativ gesetzt werden
     IF #sbOff1 AND #sbReady AND #sbIOp AND NOT #sbFault THEN

       // Tippen positiv
       IF #Jog1 AND NOT #Jog2 THEN
         //#sxSendBuf.sxSTW1.Jog1 := True;
         #sxSendBuf.STW1.%X8 := True;
       END_IF;

       // Tippen negativ
       IF #Jog2 AND NOT #Jog1 THEN
         //#sxSendBuf.sxSTW1.Jog2 := True;
         #sxSendBuf.STW1.%X9 := True;
       END_IF;

       // "Fliegendes Referentieren" aktivieren
       // "Fliegendes Referenzieren" erst nach Einschalten des Antriebes möglich
       IF #sbRefTyp THEN

         // Referenziertyp auf "Fliegendes Referenzieren" einstellen
         //#sxSendBuf.sxEPosSTW2.RefTyp := #FlyRef;
         #sxSendBuf.EPosSTW2.%X8 := #FlyRef;

         // Nach der Anwahl des Referenziertyps "Fliegendes Referenzieren", 
         // ein Zyklus später kann das Referenzieren gestartet
         IF (#siRefTypCyc = 0) THEN
           #siRefTypCyc := #siRefTypCyc + 1;
         ELSE
           // Referenzieren starten
           //#sxSendBuf.sxSTW1.RefStart := True;
           #sxSendBuf.STW1.%X11 := True;
         END_IF;
       END_IF;
     END_IF;

     // Betriebsart "Tippen positiv / Tippen negativ inkrementell" 
   ELSIF #siModePos = 8 AND #sbModePos THEN

     // Antrieb einschalten
     //#sxSendBuf.sxSTW1.OFF1 := #sbOff1;
     #sxSendBuf.STW1.%X0 := #sbOff1;

     // nicht verwendete Signale für den 1. Schritt und eventuell weitere Schritte
     (*#sxSendBuf.sxEPosSTW1.MdiStart := False;
             #sxSendBuf.sxEPosSTW2.JogInc   := False;
             #sxSendBuf.sxSTW1.Jog1         := False;
             #sxSendBuf.sxSTW1.Jog2         := False;
             #sxSendBuf.sxSTW1.RefStart     := False;
             #sxSendBuf.sxEPosSTW2.RefTyp   := False;*)

     #sxSendBuf.EPosSTW1.%X15 := False;
     #sxSendBuf.EPosSTW2.%X5 := False;
     #sxSendBuf.STW1.%X8 := False;
     #sxSendBuf.STW1.%X9 := False;
     #sxSendBuf.STW1.%X11 := False;
     #sxSendBuf.EPosSTW2.%X8 := False;

     // Nach dem Einschalten des Antriebes, ein Paar Zyklen warten bevor Tippen negativ gesetzt werden kann
     // Nach dem Einschalten des Antriebes, prüfen ob der Antrieb betriebsbereit, in Operation ohne Fehler und Warnung ist, 
     // dann kann Tippen positiv oder negativ gesetzt werden
     IF #sbOff1 AND #sbReady AND #sbIOp AND NOT #sbFault THEN

       // Tippen inkrementell einstellen
       //#sxSendBuf.sxEPosSTW2.JogInc := True;
       #sxSendBuf.EPosSTW2.%X5 := True;

       #sbJogInc := True;

       // Nach dem Einstellen des Antriebes, ein Paar Zyklen warten bevor Tippen negativ oder Tippen positiv gesetz werden kann
       IF #sbJogInc AND (#siJogIncCyc = 0) THEN
         #siJogIncCyc := #siJogIncCyc + 1;
       ELSE

         // Tippen positiv oder negativ inkrementell zulassen
         IF #Jog1 XOR #Jog2 THEN

           //#sxSendBuf.sxSTW1.Jog1 := #Jog1;
           //#sxSendBuf.sxSTW1.Jog2 := #Jog2;
           #sxSendBuf.STW1.%X8 := #Jog1;
           #sxSendBuf.STW1.%X9 := #Jog2;
         END_IF;
       END_IF;

       // "Fliegendes Referentieren" aktivieren
       // "Fliegendes Referenzieren" erst nach Einschalten des Antriebes möglich
       IF #sbRefTyp THEN

         // Referenziertyp auf "Fliegendes Referenzieren" einstellen
         //#sxSendBuf.sxEPosSTW2.RefTyp := True;
         #sxSendBuf.EPosSTW2.%X8 := True;

         // Nach der Anwahl des Referenziertyps "Fliegendes Referenzieren", 
         // ein Zyklus später kann das Referenzieren gestartet
         IF (#siRefTypCyc = 0) THEN
           #siRefTypCyc := #siRefTypCyc + 1;
         ELSE
           // Referenzieren starten
           //#sxSendBuf.sxSTW1.RefStart := True;
           #sxSendBuf.STW1.%X11 := True;
         END_IF;
       END_IF;
     END_IF;
   ELSE
     // Werte wieder zurücknehmen
     (*#sxSendBuf.sxSTW1.Off1          := #Off1;
             #sxSendBuf.sxSTW1.RejTrvTsk     := False;
             #sxSendBuf.sxSTW1.TrvStart      := False;
             #sxSendBuf.sxEPosSTW1.MdiStart  := False;
             #sxSendBuf.sxSTW1.Jog1          := False;
             #sxSendBuf.sxSTW1.Jog2          := False;
             #sxSendBuf.sxEPosSTW1.MdiTyp    := False;
             #sxSendBuf.sxEPosSTW1.MdiPos    := False;
             #sxSendBuf.sxEPosSTW1.MdiNeg    := False;
             #sxSendBuf.sxEPosSTW1.MdiTrTyp  := False;
             #sxSendBuf.sxEPosSTW1.MdiSetup  := False;
             #sxSendBuf.sxEPosSTW2.SetRefPt  := False;
             #sxSendBuf.sxEPosSTW2.RefTyp    := False;
             #sxSendBuf.sxEPosSTW2.RefStDi   := False;
             #sxSendBuf.sxEPosSTW2.JogInc    := False;
             #sxSendBuf.sxSTW1.RefStart      := False;*)

     #sxSendBuf.STW1.%X0 := #EnableAxis;
     #sxSendBuf.STW1.%X4 := False;
     #sxSendBuf.STW1.%X6 := False;
     #sxSendBuf.EPosSTW1.%X15 := False;
     #sxSendBuf.STW1.%X8 := False;
     #sxSendBuf.STW1.%X9 := False;
     #sxSendBuf.EPosSTW1.%X8 := False;
     #sxSendBuf.EPosSTW1.%X9 := False;
     #sxSendBuf.EPosSTW1.%X10 := False;
     #sxSendBuf.EPosSTW1.%X12 := False;
     #sxSendBuf.EPosSTW1.%X14 := False;
     #sxSendBuf.EPosSTW2.%X1 := False;
     #sxSendBuf.EPosSTW2.%X8 := False;
     #sxSendBuf.EPosSTW2.%X9 := False;
     #sxSendBuf.EPosSTW2.%X5 := False;
     #sxSendBuf.STW1.%X11 := False;
   END_IF; // Hauptbetriebsart "Verfahrsätze" (Traversing Blocks)

   //Den Eingang ConfigEPos auf die einzelnen Bits im Telegramm verschalten
   #sxSendBuf.STW1.%X1 := #ConfigEPos.%X0;
   #sxSendBuf.STW1.%X2 := #ConfigEPos.%X1;
   #sxSendBuf.EPosSTW2.%X14 := #ConfigEPos.%X2;
   #sxSendBuf.EPosSTW2.%X15 := #ConfigEPos.%X3;
   #sxSendBuf.EPosSTW2.%X11 := #ConfigEPos.%X4;
   #sxSendBuf.EPosSTW2.%X10 := #ConfigEPos.%X5;
   #sxSendBuf.EPosSTW2.%X2 := #ConfigEPos.%X6;
   #sxSendBuf.STW1.%X13 := #ConfigEPos.%X7;
   #sxSendBuf.EPosSTW1.%X12 := #ConfigEPos.%X8;
   #sxSendBuf.STW2.%X0 := #ConfigEPos.%X9;
   #sxSendBuf.STW2.%X1 := #ConfigEPos.%X10;
   #sxSendBuf.STW2.%X2 := #ConfigEPos.%X11;
   #sxSendBuf.STW2.%X3 := #ConfigEPos.%X12;
   #sxSendBuf.STW2.%X4 := #ConfigEPos.%X13;
   #sxSendBuf.STW2.%X7 := #ConfigEPos.%X14;
   #sxSendBuf.STW1.%X12 := #ConfigEPos.%X15;
   #sxSendBuf.STW1.%X14 := #ConfigEPos.%X16;
   #sxSendBuf.STW1.%X15 := #ConfigEPos.%X17;
   #sxSendBuf.EPosSTW1.%X6 := #ConfigEPos.%X18;
   #sxSendBuf.EPosSTW1.%X7 := #ConfigEPos.%X19;
   #sxSendBuf.EPosSTW1.%X11 := #ConfigEPos.%X20;
   #sxSendBuf.EPosSTW1.%X13 := #ConfigEPos.%X21;
   #sxSendBuf.EPosSTW2.%X3 := #ConfigEPos.%X22;
   #sxSendBuf.EPosSTW2.%X4 := #ConfigEPos.%X23;
   #sxSendBuf.EPosSTW2.%X6 := #ConfigEPos.%X24;
   #sxSendBuf.EPosSTW2.%X7 := #ConfigEPos.%X25;
   #sxSendBuf.EPosSTW2.%X12 := #ConfigEPos.%X26;
   #sxSendBuf.EPosSTW2.%X13 := #ConfigEPos.%X27;
   #sxSendBuf.STW2.%X5 := #ConfigEPos.%X28;
   #sxSendBuf.STW2.%X6 := #ConfigEPos.%X29;
   #sxSendBuf.STW2.%X8 := #ConfigEPos.%X30;
   #sxSendBuf.STW2.%X9 := #ConfigEPos.%X31;


   #swSendBuf[0] := #sxSendBuf.STW1;
   #swSendBuf[1] := #sxSendBuf.EPosSTW1;
   #swSendBuf[2] := #sxSendBuf.EPosSTW2;
   #swSendBuf[3] := #sxSendBuf.STW2;
   #swSendBuf[4] := #sxSendBuf.OverrideV;
   #swSendBuf[5] := #sxSendBuf.Position.%W1;
   #swSendBuf[6] := #sxSendBuf.Position.%W0;
   #swSendBuf[7] := #sxSendBuf.Velocity.%W1;
   #swSendBuf[8] := #sxSendBuf.Velocity.%W0;
   #swSendBuf[9] := #sxSendBuf.OverrideA;
   #swSendBuf[10] := #sxSendBuf.OverrideD;
   #swSendBuf[11] := #sxSendBuf.Reserve;

   //Prozessdaten zur Signalbaugruppe schreiben
   #piRetSFC := DPWR_DAT(LADDR := #HWIDSTW,
                         RECORD := #swSendBuf);

   // Fehler der Rückmeldung ausgeben
   #DiagID := INT_TO_WORD(#piRetSFC);

   //kein Fehler beim Schreiben
   IF #piRetSFC = 0 THEN

       // Fehler wieder zurück nehmen
       IF (#swStatus = 16#8601) THEN
           #swStatus := 16#7002;
           #Error := False;
       END_IF;

       //Prozessdaten von der Signalbaugruppe lesen
       #piRetSFC := DPRD_DAT(LADDR := #HWIDZSW,
                             RECORD => #swRecvBuf);

       // Fehlermeldung der Rückmeldung ausgeben
       #DiagID := INT_TO_WORD(#piRetSFC);

       //Fehler beim Lesen (Profibus-Kommunikation unterbrochen)
       IF #piRetSFC <> 0 THEN

           // Fehler
           #Error := TRUE;
           #swStatus := 16#8600;

           // Zustandsworte löschen
           #sxRecvBuf.ZSW1 := W#16#0;
           #sxRecvBuf.EPosZSW1 := W#16#0;
           #sxRecvBuf.EPosZSW2 := W#16#0;
           #sxRecvBuf.ZSW2 := W#16#0;
           #sxRecvBuf.NotUsed := W#16#00;
           #sxRecvBuf.Position := DW#16#00;
           #sxRecvBuf.Velocity := DW#16#00;
           #sxRecvBuf.ErrNr := W#16#00;
           #sxRecvBuf.WarnNr := W#16#00;
           #sxRecvBuf.Reserve := W#16#00;

           // Werte auslesen
       ELSE

           // Fehler wieder zurück nehmen
           IF (#swStatus = 16#8600) THEN
               #swStatus := 16#7002;
               #Error := False;
           END_IF;

           #sxRecvBuf.ZSW1 := #swRecvBuf[0];
           #sxRecvBuf.EPosZSW1 := #swRecvBuf[1];
           #sxRecvBuf.EPosZSW2 := #swRecvBuf[2];
           #sxRecvBuf.ZSW2 := #swRecvBuf[3];
           #sxRecvBuf.NotUsed := #swRecvBuf[4];
           #sxRecvBuf.Position.%W1 := #swRecvBuf[5];
           #sxRecvBuf.Position.%W0 := #swRecvBuf[6];
           #sxRecvBuf.Velocity.%W1 := #swRecvBuf[7];
           #sxRecvBuf.Velocity.%W0 := #swRecvBuf[8];
           #sxRecvBuf.ErrNr := #swRecvBuf[9];
           #sxRecvBuf.WarnNr := #swRecvBuf[10];
           #sxRecvBuf.Reserve := #swRecvBuf[11];

           // ZSW1 aufbereiten
           //#Busy := #sxRecvBuf.sxZSW1.IOp;
           #sbBusy := #sxRecvBuf.ZSW1.%X2;

           // Fehler auswerten
       (*IF #sxRecvBuf.sxZSW1.Fault THEN
                     #ErrorId := 5;
                     #Error := True;
                 ELSIF #sxRecvBuf.sxZSW1.PowInhbt THEN 
                     #ErrorId := 6;
                     #Error := True;
                 ELSE
                     // Fehler wieder zurück nehmen
                     IF (#ErrorId = 5) OR (#ErrorId = 6) THEN
                         #ErrorId := 0;    
                         #Error := False;
                     END_IF;
                 END_IF;*)
           IF #sxRecvBuf.ZSW1.%X3 THEN
               #swStatus := 16#8401;
               #Error := True;
           ELSIF #sxRecvBuf.ZSW1.%X6 THEN
               #swStatus := 16#8402;
               #Error := True;
           ELSE
               // Fehler wieder zurück nehmen
               IF (#swStatus = 16#8401) OR (#swStatus = 16#8402) THEN
                   #swStatus := 16#7002;
                   #Error := False;
               END_IF;
           END_IF;

           // EPOS_ZSW1            
           // EPOS-Wort-1 BIT 00 --> 1 = Active traversing block bit 0
           //IF #sxRecvBuf.sxEPosZSW1.ActTrvBit0 THEN
           IF #sxRecvBuf.EPosZSW1.%X0 THEN
               #swEPosZSW1 := #swEPosZSW1 OR W#16#01;
           ELSE
               #swEPosZSW1 := #swEPosZSW1 AND W#16#FFFE;
           END_IF;

           // EPOS-Wort-1 Bit 01 --> 1 = Active traversing block bit 1
           //IF #sxRecvBuf.sxEPosZSW1.ActTrvBit1 THEN
           IF #sxRecvBuf.EPosZSW1.%X1 THEN
               #swEPosZSW1 := #swEPosZSW1 OR W#16#02;
           ELSE
               #swEPosZSW1 := #swEPosZSW1 AND W#16#FFFD;
           END_IF;

           // EPOS-Wort-1 Bit 02 --> 1 = Active traversing block bit 2
           //IF #sxRecvBuf.sxEPosZSW1.ActTrvBit2 THEN
           IF #sxRecvBuf.EPosZSW1.%X2 THEN
               #swEPosZSW1 := #swEPosZSW1 OR W#16#04;
           ELSE
               #swEPosZSW1 := #swEPosZSW1 AND W#16#FFFB;
           END_IF;

           // EPOS-Wort-1 Bit 03 --> 1 = Active traversing block bit 3
           //IF #sxRecvBuf.sxEPosZSW1.ActTrvBit3 THEN
           IF #sxRecvBuf.EPosZSW1.%X3 THEN
               #swEPosZSW1 := #swEPosZSW1 OR W#16#08;
           ELSE
               #swEPosZSW1 := #swEPosZSW1 AND W#16#FFF7;
           END_IF;

           // EPOS-Wort-1 Bit 04 --> 1 = Active traversing block bit 4 
           //IF #sxRecvBuf.sxEPosZSW1.ActTrvBit4 THEN
           IF #sxRecvBuf.EPosZSW1.%X4 THEN
               #swEPosZSW1 := #swEPosZSW1 OR W#16#10;
           ELSE
               #swEPosZSW1 := #swEPosZSW1 AND W#16#FFEF;
           END_IF;

           // EPOS-Wort-1 Bit 05 --> 1 = Active traversing block bit 5
           //IF #sxRecvBuf.sxEPosZSW1.ActTrvBit5 THEN
           IF #sxRecvBuf.EPosZSW1.%X5 THEN
               #swEPosZSW1 := #swEPosZSW1 OR W#16#20;
           ELSE
               #swEPosZSW1 := #swEPosZSW1 AND W#16#FFDF;
           END_IF;

           // EPOS-Wort-1 Bit 08 --> 1 = STOP cam minus active
           //IF #sxRecvBuf.sxEPosZSW1.StpCamMinAct THEN
           IF #sxRecvBuf.EPosZSW1.%X8 THEN
               #swEPosZSW1 := #swEPosZSW1 OR W#16#100;
           ELSE
               #swEPosZSW1 := #swEPosZSW1 AND W#16#FEFF;
           END_IF;

           // EPOS-Wort-1 Bit 09 --> 1 = STOP cam plus active
           //IF #sxRecvBuf.sxEPosZSW1.StpCamPlsAct THEN
           IF #sxRecvBuf.EPosZSW1.%X9 THEN
               #swEPosZSW1 := #swEPosZSW1 OR W#16#200;
           ELSE
               #swEPosZSW1 := #swEPosZSW1 AND W#16#FDFF;
           END_IF;

           // EPOS-Wort-1 Bit 10 --> 1 = Jogging active
           //IF #sxRecvBuf.sxEPosZSW1.JogAct THEN
           IF #sxRecvBuf.EPosZSW1.%X10 THEN
               #swEPosZSW1 := #swEPosZSW1 OR W#16#400;
           ELSE
               #swEPosZSW1 := #swEPosZSW1 AND W#16#FBFF;
           END_IF;

           // EPOS-Wort-1 Bit 11 --> 1 = Reference point approach active
           //IF #sxRecvBuf.sxEPosZSW1.RefAct THEN
           IF #sxRecvBuf.EPosZSW1.%X11 THEN
               #swEPosZSW1 := #swEPosZSW1 OR W#16#800;
           ELSE
               #swEPosZSW1 := #swEPosZSW1 AND W#16#F7FF;
           END_IF;

           // Anstossen des fliegenden Referenzieren prüfen, wenn die Rückmeldung fehlt dann wiederholen
           //IF NOT #sxRecvBuf.sxEPosZSW1.FlyRefAct AND #sbRefTyp AND #sxSendBuf.sxSTW1.RefStart THEN
           IF NOT #sxRecvBuf.EPosZSW1.%X12 AND #sbRefTyp AND #sxSendBuf.STW1.%X11 THEN

               // Wiederholung anstossen 
               IF #siRefActRetry < #siRetryMax THEN
                   #siRefActRetry := #siRefActRetry + 1;

                   // Referenzieren starten wieder wegnehmen
                   //#sxSendBuf.sxSTW1.RefStart := False;
                   #sxSendBuf.STW1.%X11 := False;
               ELSE

                   // Fehlermeldung
                   #swStatus := 16#8403;
                   #Error := True;
               END_IF;
           ELSE

               // Fehler wieder zurücknehmen, wenn er mal ausgelöst wurde
               IF #swStatus = 16#8403 THEN
                   #swStatus := 16#7002;
                   #Error := False;
               END_IF;
           END_IF;

           // EPOS-Wort-1 Bit 12 --> 1 = Flying referencing active
           //IF #sxRecvBuf.sxEPosZSW1.FlyRefAct THEN
           IF #sxRecvBuf.EPosZSW1.%X12 THEN
               #swEPosZSW1 := #swEPosZSW1 OR W#16#1000;
           ELSE
               #swEPosZSW1 := #swEPosZSW1 AND W#16#EFFF;
           END_IF;

           // EPOS-Wort-1 Bit 13 --> 1 = Traversing block active
           //IF #sxRecvBuf.sxEPosZSW1.TrvBlAct THEN
           IF #sxRecvBuf.EPosZSW1.%X13 THEN
               #swEPosZSW1 := #swEPosZSW1 OR W#16#2000;
           ELSE
               #swEPosZSW1 := #swEPosZSW1 AND W#16#DFFF;
           END_IF;

           // EPOS-Wort-1 Bit 14 --> 1 = MDI setup active
           //IF #sxRecvBuf.sxEPosZSW1.MdiStupAct THEN
           IF #sxRecvBuf.EPosZSW1.%X14 THEN
               #swEPosZSW1 := #swEPosZSW1 OR W#16#4000;
           ELSE
               #swEPosZSW1 := #swEPosZSW1 AND W#16#BFFF;
           END_IF;

           // EPOS-Wort-1 Bit 15 --> 1 = MDI positing active
           //IF #sxRecvBuf.sxEPosZSW1.MdiPosAct THEN
           IF #sxRecvBuf.EPosZSW1.%X15 THEN
               #swEPosZSW1 := #swEPosZSW1 OR W#16#8000;
           ELSE
               #swEPosZSW1 := #swEPosZSW1 AND W#16#7FFF;
           END_IF;

           // EPOS_ZSW2 
           // EPOS-Wort-2 Bit 00 --> 1 = Tracking mode active
           //IF #sxRecvBuf.sxEPosZSW2.TrkModeAct THEN
           IF #sxRecvBuf.EPosZSW2.%X0 THEN
               #swEPosZSW2 := #swEPosZSW2 OR W#16#01;
           ELSE
               #swEPosZSW2 := #swEPosZSW2 AND W#16#FFFE;
           END_IF;

           // EPOS-Wort-2 Bit 01 --> 1 = Velocity limit active
           //IF #sxRecvBuf.sxEPosZSW2.VeloLimAct THEN
           IF #sxRecvBuf.EPosZSW2.%X1 THEN
               #swEPosZSW2 := #swEPosZSW2 OR W#16#02;
           ELSE
               #swEPosZSW2 := #swEPosZSW2 AND W#16#FFFD;
           END_IF;

           // EPOS-Wort-2 Bit 02 --> 1 = Setpoint static
           //IF #sxRecvBuf.sxEPosZSW2.SetPStat THEN
           IF #sxRecvBuf.EPosZSW2.%X2 THEN
               #swEPosZSW2 := #swEPosZSW2 OR W#16#04;
           ELSE
               #swEPosZSW2 := #swEPosZSW2 AND W#16#FFFB;
           END_IF;

           // EPOS-Wort-2 Bit 03 --> 1 = Printmark outside outer window
           //IF #sxRecvBuf.sxEPosZSW2.PrnMrkOut THEN
           IF #sxRecvBuf.EPosZSW2.%X3 THEN
               #swEPosZSW2 := #swEPosZSW2 OR W#16#08;
           ELSE
               #swEPosZSW2 := #swEPosZSW2 AND W#16#FFF7;
           END_IF;

           // EPOS-Wort-2 Bit 04 --> 1 = Axis forwards
           //IF #sxRecvBuf.sxEPosZSW2.FWD THEN
           IF #sxRecvBuf.EPosZSW2.%X4 THEN
               #swEPosZSW2 := #swEPosZSW2 OR W#16#10;
           ELSE
               #swEPosZSW2 := #swEPosZSW2 AND W#16#FFEF;
           END_IF;

           // EPOS-Wort-2 Bit 05 --> 1 = Axis backwards
           //IF #sxRecvBuf.sxEPosZSW2.BWD THEN
           IF #sxRecvBuf.EPosZSW2.%X5 THEN
               #swEPosZSW2 := #swEPosZSW2 OR W#16#20;
           ELSE
               #swEPosZSW2 := #swEPosZSW2 AND W#16#FFDF;
           END_IF;

           // EPOS-Wort-2 Bit 06 --> 1 = Software limit switch minus active
           //IF #sxRecvBuf.sxEPosZSW2.SftSwMinAct THEN
           IF #sxRecvBuf.EPosZSW2.%X6 THEN
               #swEPosZSW2 := #swEPosZSW2 OR W#16#40;
           ELSE
               #swEPosZSW2 := #swEPosZSW2 AND W#16#FFBF;
           END_IF;

           // EPOS-Wort-2 Bit 07 --> 1 = Software limit switch plus active
           //IF #sxRecvBuf.sxEPosZSW2.SftSwPlsAct THEN
           IF #sxRecvBuf.EPosZSW2.%X7 THEN
               #swEPosZSW2 := #swEPosZSW2 OR W#16#80;
           ELSE
               #swEPosZSW2 := #swEPosZSW2 AND W#16#FF7F;
           END_IF;

           // EPOS-Wort-2 Bit 08 --> 1 = Position actual value <= cam position 1
           //IF #sxRecvBuf.sxEPosZSW2.PosSmCam1 THEN
           IF #sxRecvBuf.EPosZSW2.%X8 THEN
               #swEPosZSW2 := #swEPosZSW2 OR W#16#100;
           ELSE
               #swEPosZSW2 := #swEPosZSW2 AND W#16#FEFF;
           END_IF;

           // EPOS-Wort-2 Bit 09 --> 1 = Position actual value <= cam position 2
           //IF #sxRecvBuf.sxEPosZSW2.PosSmCam2 THEN
           IF #sxRecvBuf.EPosZSW2.%X9 THEN
               #swEPosZSW2 := #swEPosZSW2 OR W#16#200;
           ELSE
               #swEPosZSW2 := #swEPosZSW2 AND W#16#FDFF;
           END_IF;

           // EPOS-Wort-2 Bit 10 --> 1 = Direct output 1 via traversing block
           //IF #sxRecvBuf.sxEPosZSW2.TrvOut1 THEN
           IF #sxRecvBuf.EPosZSW2.%X10 THEN
               #swEPosZSW2 := #swEPosZSW2 OR W#16#400;
           ELSE
               #swEPosZSW2 := #swEPosZSW2 AND W#16#FBFF;
           END_IF;

           // EPOS-Wort-2 Bit 11 --> 1 = Direct output 2 via traversing block
           //IF #sxRecvBuf.sxEPosZSW2.TrvOut2 THEN
           IF #sxRecvBuf.EPosZSW2.%X11 THEN
               #swEPosZSW2 := #swEPosZSW2 OR W#16#800;
           ELSE
               #swEPosZSW2 := #swEPosZSW2 AND W#16#F7FF;
           END_IF;

           // EPOS-Wort-2 Bit 12 --> 1 = Fixed STOP reached
           //IF #sxRecvBuf.sxEPosZSW2.FxStpRd THEN
           IF #sxRecvBuf.EPosZSW2.%X12 THEN
               #swEPosZSW2 := #swEPosZSW2 OR W#16#1000;
           ELSE
               #swEPosZSW2 := #swEPosZSW2 AND W#16#EFFF;
           END_IF;

           // EPOS-Wort-2 Bit 13 --> 1 = Fixed STOP clamping torque reached
           //IF #sxRecvBuf.sxEPosZSW2.FxStpTrRd THEN
           IF #sxRecvBuf.EPosZSW2.%X13 THEN
               #swEPosZSW2 := #swEPosZSW2 OR W#16#2000;
           ELSE
               #swEPosZSW2 := #swEPosZSW2 AND W#16#DFFF;
           END_IF;

           // EPOS-Wort-2 Bit 14 --> 1 = Traversing fixed STOP active
           //IF #sxRecvBuf.sxEPosZSW2.TrvFxStpAct THEN
           IF #sxRecvBuf.EPosZSW2.%X14 THEN
               #swEPosZSW2 := #swEPosZSW2 OR W#16#4000;
           ELSE
               #swEPosZSW2 := #swEPosZSW2 AND W#16#BFFF;
           END_IF;

           // EPOS-Wort-2 Bit 15 --> 1 = Traversing command active
           //IF #sxRecvBuf.sxEPosZSW2.CmdAct THEN
           IF #sxRecvBuf.EPosZSW2.%X15 THEN
               #swEPosZSW2 := #swEPosZSW2 OR W#16#8000;
           ELSE
               #swEPosZSW2 := #swEPosZSW2 AND W#16#7FFF;
           END_IF;

           #sbReady := #sxRecvBuf.ZSW1.%X1;

           #AxisEnabled := #sxRecvBuf.ZSW1.%X2;
           #sbIOp := #sxRecvBuf.ZSW1.%X2;

           #AxisError := #sxRecvBuf.ZSW1.%X3;
           #sbFault := #sxRecvBuf.ZSW1.%X3;

           #AxisWarn := #sxRecvBuf.ZSW1.%X7;
           #sbAlarm := #sxRecvBuf.ZSW1.%X7;

           #AxisPosOk := #sxRecvBuf.ZSW1.%X10;
           #AxisRef := #sxRecvBuf.ZSW1.%X11;

           #sbAccel := #sxRecvBuf.ZSW1.%X14;
           #sbDecel := #sxRecvBuf.ZSW1.%X15;

           #ActVelocity := DWORD_TO_DINT(#sxRecvBuf.Velocity);
           #ActPosition := DWORD_TO_DINT(#sxRecvBuf.Position);
           #ActMode := #ModePos;
           #ActWarn := #sxRecvBuf.WarnNr;
           #ActFault := #sxRecvBuf.ErrNr;

           #Lockout := #sxRecvBuf.ZSW1.%X6;
       END_IF;
   ELSE

       // Fehler
       #Error := TRUE;
       #swStatus := 16#8601; //DPWR_DAT 错误

   END_IF;

   // Initialisierung von Ausg㭧en
   #Status := #swStatus;
   #EPosZSW1 := #swEPosZSW1;
   #EPosZSW2 := #swEPosZSW2;
END_FUNCTION_BLOCK

FUNCTION_BLOCK "SINA_PARA_S"   // FB1821, SCL
{ S7_Optimized_Access := 'TRUE' }
AUTHOR : DRVDPS7
FAMILY : DRIVES
NAME : SINA_PAS
VERSION : 5.0
// stored: AutoNumber false, MemoryReserve 100, SetENOAutomatically false
   VAR_INPUT
      Start : Bool := 0;
      ReadWrite : Bool := 0;
      Parameter : Int := 1;
      Index : Int := 0;
      ValueWrite1 : Real := 0.0;
      ValueWrite2 : DInt := 0;
      AxisNo : Byte := 16#01;
      hardwareId : HW_IO := 0;
   END_VAR
   VAR_OUTPUT
      Ready : Bool := 0;
      Busy : Bool := 0;
      Done : Bool := 1;
      ValueRead1 : Real := 0.0;
      ValueRead2 : DInt := 0;
      Format : Byte := 16#00;
      ErrorNo : Word := 16#0000;
      Error : Bool := 0;
      ErrorId : DWord := 0;
      DiagId : Word := 16#0000;
   END_VAR
   VAR
      sbWrError : Bool := 0;
      sbWrDone : Bool := 0;
      sbRdError : Bool := 0;
      sbWrBusy : Bool := 0;
      sbRdBusy : Bool := 0;
      sbWrStart : Bool := 0;
      sbRdStart : Bool := 0;
      sbWrStart1 : Bool := 0;
      sbRdStart1 : Bool := 0;
      sbWrStart2 : Bool := 0;
      sbRdStart2 : Bool := 0;
      sbStart : Bool := 0;
      sbReady : Bool := 0;
      sbRead : Bool := 0;
      sbWrite : Bool := 0;
      sbParaNo : Bool := 0;
      sbBusy : Bool := 0;
      sbError : Bool := 0;
      sbDone : Bool := 0;
      syFormat : Byte := 16#00;
      syAxisNo : Byte := 0;
      siReqRef : Int := 0;
      siErrorId : Int := 0;
      siErrorCount : Int := 0;
      siMaxErrCount : Int := 12500;
      swParaError : Word := WORD#16#0000;
      sxReqParaMulti : Struct
         sxHeader : Struct
            syReqRef : Byte := 16#00;
            syReqId : Byte := 16#01;
            syAxisNo : Byte := 16#00;
            syParaNo : Byte := 16#00;
         END_STRUCT;
         sxParaAdress : Struct
            syAttr : Byte := 16#10;
            syElemNo : Byte := 16#01;
            siParaNo : Int := 0;
            siIndex : Int := 0;
         END_STRUCT;
      END_STRUCT;
      sxChaParaMulti : Struct
         sxHeader : Struct
            syReqRef : Byte := 16#00;
            syReqId : Byte := 16#02;
            syAxisNo : Byte := 16#00;
            syParaNo : Byte := 16#00;
         END_STRUCT;
         sxData : Array[1..12] of Byte;
      END_STRUCT;
      sxRespParaMulti : Struct
         sxHeader : Struct
            syReqRef : Byte := 16#00;
            syReqId : Byte := 16#00;
            syAxisNo : Byte := 16#00;
            syParaNo : Byte := 16#00;
         END_STRUCT;
         sxData : Array[1..6] of Byte;
      END_STRUCT;
      RDREC_1 { S7_SetPoint := 'True'} : RDREC;
      WRREC_1 { S7_SetPoint := 'True'} : WRREC;
      siLenHeader : Int := 4;
      siLenParaMulti : Int := 6;
      siLenChaPara : Int := 12;
   END_VAR
   VAR_TEMP
      piCount : Int;
      piPointer : Int;
      piLenTele : Int;
      piRetSFC : Int;
      pwWordHigh : Word;
      pwWordLow : Word;
      pwWord1 : Word;
      pwWord2 : Word;
      pdDWordHigh : DWord;
      pdDWordLow : DWord;
      pdStatus : DWord;
      pbValidSFB : Bool;
      piLenSFB : UInt;
      pwErrorNo : Word;
   END_VAR
BEGIN

   //=============================================================================
   //SIEMENS AG
   //(c)Copyright 2017 All Rights Reserved
   //-----------------------------------------------------------------------------
   // Library: DriveLib
   // Tested with: S7-1516-3 PN/DP V1.8
   // Engineering: TIA Portal V14
   // Restrictions: -
   // Requirements: S7-1200 / S7-1500
   // Functionality: read and write one parameter from/to a Sinamics
   //
   //=============================================================================

   // Auftrag "Parameter lesen" bzw. Auftrag "Parameter schreiben" wird nicht mehr ausgeführt
   IF NOT #sbBusy THEN
     #sbParaNo := TRUE;
     #syAxisNo := #AxisNo;
   END_IF;

   // Starten 
   IF #Start AND NOT #sbStart AND NOT #sbBusy THEN

     #sbReady := False;
     #sbError := False;
     #sbBusy := False;

     // Auftrag "Parameter lesen" erkennen
     IF NOT #ReadWrite THEN
       #sbRead := True;
       #sbWrStart := True;
       #sbRdStart := False;

       #sbWrite := False;
       #sbWrStart1 := False;
       #sbRdStart1 := False;
       #sbWrStart2 := False;
       #sbRdStart2 := False;

       // Referenzauftragsnummer erzeugen
       #siReqRef := #siReqRef + 1;

       // bei Überschreitung wieder zurücksetzen und von vorne (Wertebereich von 0-255)
       IF #siReqRef > 255 THEN
         #siReqRef := 0;
       END_IF;

       // Auftrag "Parameter schreiben" erkennen
     ELSE
       #sbWrite := True;
       #sbWrStart1 := True;
       #sbRdStart1 := False;
       #sbWrStart2 := False;
       #sbRdStart2 := False;

       #sbRead := False;
       #sbWrStart := False;
       #sbRdStart := False;

       // Referenzauftragsnummer erzeugen
       #siReqRef := #siReqRef + 1;

       // bei Überschreitung wieder zurücksetzen und von vorne (Wertebereich von 0-255)
       IF #siReqRef > 255 THEN
         #siReqRef := 0;
       END_IF;
     END_IF;

     // Fehler 4 und 5 wieder zurücknehmen
     IF (#siErrorId = 4) OR (#siErrorId = 5) THEN
       #sbError := False;
       #siErrorId := 0;
     END_IF;
   END_IF;

   // "Start commando" Flanke merken
   #sbStart := #Start;

   // Abbrechen
   IF NOT #Start THEN

     #siErrorCount := 0;
     // Schreib - oder Lesevorgang abbrechen
     #sbRead := False;
     #sbWrStart := False;
     #sbRdStart := False;

     #sbWrite := False;
     #sbWrStart1 := False;
     #sbRdStart1 := False;
     #sbWrStart2 := False;
     #sbRdStart2 := False;

     // Auftag ist noch beschäftigt => Fehler ausgeben
     IF #sbBusy THEN
       #sbError := True;
       #siErrorId := 4;
       #sbBusy := False;
     END_IF;
   END_IF;


   // Auftrag "Parameter lesen" wurde ausgelöst
   IF #sbParaNo AND #sbRead AND NOT #sbWrite THEN

     // Auftrag "Parameter lesen" vorbereiten und abschicken
     IF #sbWrStart THEN

       // Ablöschen des Sendepuffers
       // Parameternummer des Parameters 
       #sxReqParaMulti.sxParaAdress.siParaNo := 0;

       // Subindex des Parameters
       #sxReqParaMulti.sxParaAdress.siIndex := 0;

       // Auftrags-HEADER erstellen
       // Auftragsreferenz
       #sxReqParaMulti.sxHeader.syReqRef := INT_TO_BYTE(#siReqRef);

       // Auftragskennung 0x01=Request Parameters
       #sxReqParaMulti.sxHeader.syReqId := B#16#01;

       // Achse
       #sxReqParaMulti.sxHeader.syAxisNo := #syAxisNo;

       // Anzahl Parameter        
       #sxReqParaMulti.sxHeader.syParaNo := B#16#01;

       // Auftrags-PARAMETERADRESSE erstellen
       // Parameternummer des Parameters                                
       #sxReqParaMulti.sxParaAdress.siParaNo := #Parameter;

       // Subindex des Parameters
       #sxReqParaMulti.sxParaAdress.siIndex := #Index;

       // SCHREIBEN AZYKLISCH
       #piLenTele := #siLenHeader + #siLenParaMulti;
       #WRREC_1(REQ := True,                                // Startimpuls
                ID := #hardwareId,                         // Diagnoseadresse
                INDEX := 47,                                  // Rahmentyp
                LEN := INT_TO_UINT(#piLenTele),             // maximale Länge
                DONE => #sbWrDone,                           // Schreibauftrag beendet
                BUSY => #sbWrBusy,                           // Slave beschäftigt
                ERROR => #sbWrError,                          // Fehler beim Schreiben
                STATUS => #pdStatus,                           // Status[1] = Error => Status[2] Error Decode + Status[3] Error Code
                RECORD := #sxReqParaMulti);                    // Zeiger auf zu schreibenen Datensatzes

       // Ausgänge setzen
       #sbBusy := #sbWrBusy;
       #sbDone := #sbWrDone;

       // Fehler auswerten
       IF #sbWrError THEN

         // Fehlerstatus aus dem Doppelwort filtern und weitergeben                
         #pwWord1 := DWORD_TO_WORD(SHR(IN := (#pdStatus AND DW#16#FFFF00), N := 8));

         // Fehlerstatus setzen
         #siErrorId := 3;
         #DiagId := #pwWord1;

         //Temporärer Fehler: #pdStatus = 80A7, 80B5, 80C0, 80C1, 80C2, 80C3 oder 80C4 zulassen und nocheinmal versuchen
         IF NOT (#pwWord1 = DW#16#80A7) AND NOT (#pwWord1 = DW#16#80B5) AND NOT (#pwWord1 = DW#16#80C0) AND
           NOT (#pwWord1 = DW#16#80C1) AND NOT (#pwWord1 = DW#16#80C2) AND NOT (#pwWord1 = DW#16#80C3) AND
           NOT (#pwWord1 = DW#16#80C4) THEN

           // Wiederholungsauftrag wieder zurücknehmen 
           #sbWrStart := False;
           #sbRdStart := False;
           #sbRead := False;

           // Fehler ausgeben 
           #sbError := #sbWrError;

         ELSE
           // Fehlerwiederholauftrag ??                   
           IF #siErrorCount = #siMaxErrCount THEN

             // Wiederholungsauftrag wieder zurücknehmen
             #sbWrStart := False;
             #sbRdStart := False;
             #sbRead := False;

             //Fehlerzähler zurücksetzen
             #siErrorCount := 0;


             // Fehler ausgeben 
             #sbError := #sbWrError;

             // nix tun bis Zähler überläuft
           ELSE
             #siErrorCount := #siErrorCount + 1;
           END_IF;
         END_IF;

         // kein Fehler beim SCHEIBEN AZYKLISCH und Auftrag fertig 
       ELSIF NOT #sbWrBusy AND #sbWrDone THEN

         // Fehlerkennung zurücknehmen
         IF #siErrorId = 3 THEN
           #siErrorId := 0;
           #sbError := False;
         END_IF;

         #DiagId := W#16#00;

         // Schreibauftrag fertig melden und Leseantrag anstossen
         #sbWrStart := False;
         #sbRdStart := True;
       END_IF;
     END_IF; // Auftrag "Parameter lesen" vorbereiten und abschicken

     // vom Auftrag "Parameter lesen" die Antwort abwarten und dann auswerten
     IF #sbRdStart THEN

       // Ablöschen des Empfangspuffers
       #sxRespParaMulti.sxHeader.syReqRef := B#16#00;
       #sxRespParaMulti.sxHeader.syReqId := B#16#00;
       #sxRespParaMulti.sxHeader.syAxisNo := B#16#00;
       #sxRespParaMulti.sxHeader.syParaNo := B#16#00;

       FOR #piCount := 1 TO #siLenParaMulti DO
         #sxRespParaMulti.sxData[#piCount] := B#16#00;
       END_FOR;

       // LESEN AZYKLISCH
       #piLenTele := #siLenHeader + #siLenParaMulti;
       #RDREC_1(REQ := True,                                // Startimpuls
                ID := #hardwareId,                         // Diagnoseadresse        
                INDEX := 47,                                  // Rahmentyp           
                MLEN := INT_TO_UINT(#piLenTele),             // maximale Länge
                VALID => #pbValidSFB,                         // neuer Datensatz empfangen und gültig   
                BUSY => #sbRdBusy,                           // Slave beschäftigt
                ERROR => #sbRdError,                          // Fehler beim Schreiben
                STATUS => #pdStatus,                           // Status[1] = Error => Status[2] Error Decode + Status[3] Error Code 
                LEN => #piLenSFB,                           // Länge des gelesenen Datensatzes
                RECORD := #sxRespParaMulti);                   // Zeiger auf gelesenen Datensatz

       // Ausgänge setzen
       #sbBusy := #sbRdBusy;
       #sbDone := #pbValidSFB;

       // Fehler auswerten
       IF #sbRdError THEN
         // Fehlerstatus aus dem Doppelwort filtern und weitergeben                
         #pwWord1 := DWORD_TO_WORD(SHR(IN := (#pdStatus AND DW#16#FFFF00), N := 8));

         // Fehlerstatus setzen
         #siErrorId := 3;
         #DiagId := #pwWord1;

         //Temporärer Fehler: #pdStatus = 80A7, 80B5, 80C0, 80C1, 80C2, 80C3 oder 80C4 zulassen und nocheinmal versuchen
         IF NOT (#pwWord1 = DW#16#80A7) AND NOT (#pwWord1 = DW#16#80B5) AND NOT (#pwWord1 = DW#16#80C0) AND
           NOT (#pwWord1 = DW#16#80C1) AND NOT (#pwWord1 = DW#16#80C2) AND NOT (#pwWord1 = DW#16#80C3) AND
           NOT (#pwWord1 = DW#16#80C4) THEN

           // Wiederholungsauftrag wieder zurücknehmen  
           #sbWrStart := False;
           #sbRdStart := False;
           #sbRead := False;

           // Fehler ausgeben 
           #sbError := #sbRdError;

         ELSE
           // Fehlerwiederholauftrag ??                   
           IF #siErrorCount = #siMaxErrCount THEN

             // Wiederholungsauftrag wieder zurücknehmen
             #sbWrStart := False;
             #sbRdStart := False;
             #sbRead := False;

             //Fehlerzähler zurücksetzen
             #siErrorCount := 0;


             // Fehler ausgeben 
             #sbError := #sbRdError;

             // nix tun bis Zähler überläuft
           ELSE
             #siErrorCount := #siErrorCount + 1;
           END_IF;
         END_IF;

         // Fehler : die Auftragsreferenz der Antwort übertimmt nicht mit der Auftragsreferenz der Anfrage überein
       ELSIF NOT (#siReqRef = BYTE_TO_INT(#sxRespParaMulti.sxHeader.syReqRef)) AND NOT #sbRdBusy AND #pbValidSFB THEN
         #siErrorId := 1;
         #sbError := True;
         #sbDone := False;

         // Wiederholungsauftrag wieder zurücknehmen  
         #sbWrStart := False;
         #sbRdStart := False;
         #sbRead := False;

         // Fehler : falsche Auftragskennung zurück erhalten    
       ELSIF NOT (#sxRespParaMulti.sxHeader.syReqId = B#16#81 OR #sxRespParaMulti.sxHeader.syReqId = B#16#01) AND
         NOT #sbRdBusy AND #pbValidSFB THEN
         #siErrorId := 1;
         #sbError := True;
         #sbDone := False;

         // Wiederholungsauftrag wieder zurücknehmen  
         #sbWrStart := False;
         #sbRdStart := False;
         #sbRead := False;

         // Fehler : die angeforderte Anzahl Parameter entspricht nicht der übermittelten Anzahl Parameter überein
       ELSIF NOT (#sxRespParaMulti.sxHeader.syParaNo = B#16#01) AND NOT #sbRdBusy AND #pbValidSFB THEN
         #siErrorId := 1;
         #sbError := True;
         #sbDone := False;

         // Wiederholungsauftrag wieder zurücknehmen  
         #sbWrStart := False;
         #sbRdStart := False;
         #sbRead := False;

         // Fehler : die Achse entspricht nicht der übergebenen Achse
       ELSIF NOT (#syAxisNo = #sxRespParaMulti.sxHeader.syAxisNo) AND NOT #sbRdBusy AND #pbValidSFB THEN
         #siErrorId := 1;
         #sbError := True;
         #sbDone := False;

         // Wiederholungsauftrag wieder zurücknehmen  
         #sbWrStart := False;
         #sbRdStart := False;
         #sbRead := False;

         // kein Fehler beim LESEN AZYKLISCH und Auftrag fertig 
       ELSIF NOT #sbRdBusy AND #pbValidSFB THEN

         // die angefragten Parameter auswerten und im Puffer abspeichern

         // ermitteltes Format des Parameters abspeichern
         #syFormat := #sxRespParaMulti.sxData[1];

         // Format = Error ? = > gesendeter Parameter fehlerhaft
         IF (BYTE_TO_INT(#sxRespParaMulti.sxData[1]) = 68) THEN

           // Format = Error, zwei Bytes zu übermittelten Fehlernummer zusammenfassen
           #pwWordHigh := SHL(IN := BYTE_TO_WORD(#sxRespParaMulti.sxData[3]), N := 8);
           #pwWordLow := BYTE_TO_WORD(#sxRespParaMulti.sxData[4]);

           #sbError := True;

           // ermittelte Fehlernummer im Puffer abspeichern
           #ErrorNo := #pwWordHigh XOR #pwWordLow;

           // Die Fehlerhaftigkeit des erkannten Parameter in der Fehlernummer eintragen   
           #swParaError := #swParaError OR W#16#01;

           // Format = Byte ? = > gesendeter Parameter ein Byte lang ohne Vorzeichen
         ELSIF (#sxRespParaMulti.sxData[1] = B#16#41) OR (#sxRespParaMulti.sxData[1] = B#16#05) THEN

           // ermittelter Parameterwert eintragen (Byte) 
           #ValueRead1 := USINT_TO_REAL(BYTE_TO_USINT(#sxRespParaMulti.sxData[3]));
           #ValueRead2 := 0;

           // ermittelte Fehlernummer im Puffer zurücksetzen
           #ErrorNo := W#16#00;

           // Die Fehlerhaftigkeit des erkannten Parameter in der Fehlernummer löschen   
           #swParaError := #swParaError AND W#16#FFFE;

           // Format = Byte ? = > gesendeter Parameter ein Byte lang mit Vorzeichen
         ELSIF (#sxRespParaMulti.sxData[1] = B#16#02) THEN

           // ermittelter Parameterwert eintragen (Byte) 
           #ValueRead1 := SINT_TO_REAL(BYTE_TO_SINT(#sxRespParaMulti.sxData[3]));
           #ValueRead2 := 0;

           // ermittelte Fehlernummer im Puffer zurücksetzen
           #ErrorNo := W#16#00;

           // Die Fehlerhaftigkeit des erkannten Parameter in der Fehlernummer löschen   
           #swParaError := #swParaError AND W#16#FFFE;

           // Format = Word ? = > gesendeter Parameter zwei Bytes lang ohne Vorzeichen
         ELSIF (#sxRespParaMulti.sxData[1] = B#16#42) OR (#sxRespParaMulti.sxData[1] = B#16#06)
           OR (#sxRespParaMulti.sxData[1] = B#16#0A) THEN

           // Format = Word, zwei Bytes zu übermitteltem Parameterwert zusammenfassen
           #pwWordHigh := SHL(IN := BYTE_TO_WORD(#sxRespParaMulti.sxData[3]), N := 8);
           #pwWordLow := BYTE_TO_WORD(#sxRespParaMulti.sxData[4]);
           #pwWord1 := #pwWordHigh XOR #pwWordLow;

           // ermittelter Parameterwert eintragen (Word)
           #ValueRead1 := UINT_TO_REAL(WORD_TO_UINT(#pwWord1));
           #ValueRead2 := 0;

           // ermittelte Fehlernummer im Puffer zurücksetzen
           #ErrorNo := W#16#00;

           // Die Fehlerhaftigkeit des erkannten Parameter in der Fehlernummer löschen   
           #swParaError := #swParaError AND W#16#FFFE;

           // Format = Word ? = > gesendeter Parameter zwei Bytes lang mit Vorzeichen
         ELSIF (#sxRespParaMulti.sxData[1] = B#16#03) THEN

           // Format = Word, zwei Bytes zu übermitteltem Parameterwert zusammenfassen
           #pwWordHigh := SHL(IN := BYTE_TO_WORD(#sxRespParaMulti.sxData[3]), N := 8);
           #pwWordLow := BYTE_TO_WORD(#sxRespParaMulti.sxData[4]);
           #pwWord1 := #pwWordHigh XOR #pwWordLow;

           // ermittelter Parameterwert eintragen (Word)
           #ValueRead1 := INT_TO_REAL(WORD_TO_INT(#pwWord1));
           #ValueRead2 := 0;

           // ermittelte Fehlernummer im Puffer zurücksetzen
           #ErrorNo := W#16#00;

           // Die Fehlerhaftigkeit des erkannten Parameter in der Fehlernummer löschen   
           #swParaError := #swParaError AND W#16#FFFE;

           // Format = Double Word ? = > gesendeter Parameter vier Bytes lang ohne Vorzeichen
         ELSIF (#sxRespParaMulti.sxData[1] = B#16#43) OR (#sxRespParaMulti.sxData[1] = B#16#07) OR
           (#sxRespParaMulti.sxData[1] = B#16#0D) THEN

           // Format = Double Word, vier Bytes zu übermitteltem Parameterwert zusammenfassen
           #pwWordHigh := SHL(IN := BYTE_TO_WORD(#sxRespParaMulti.sxData[3]), N := 8);
           #pwWordLow := BYTE_TO_WORD(#sxRespParaMulti.sxData[4]);
           #pwWord1 := #pwWordHigh XOR #pwWordLow;

           #pwWordHigh := SHL(IN := BYTE_TO_WORD(#sxRespParaMulti.sxData[5]), N := 8);
           #pwWordLow := BYTE_TO_WORD(#sxRespParaMulti.sxData[6]);
           #pwWord2 := #pwWordHigh XOR #pwWordLow;

           #pdDWordHigh := SHL(IN := WORD_TO_DWORD(#pwWord1), N := 16);
           #pdDWordLow := WORD_TO_DWORD(#pwWord2);

           // ermittelter Parameterwert eintragen (Word)
           #ValueRead1 := 0.0;
           #ValueRead2 := DWORD_TO_DINT(#pdDWordHigh XOR #pdDWordLow);

           // ermittelte Fehlernummer im Puffer zurücksetzen
           #ErrorNo := W#16#00;

           // Die Fehlerhaftigkeit des erkannten Parameter in der Fehlernummer löschen   
           #swParaError := #swParaError AND W#16#FFFE;

           // Format = Double Word ? = > gesendeter Parameter vier Bytes lang mit Vorzeichen
         ELSIF (#sxRespParaMulti.sxData[1] = B#16#04) THEN

           // Format = Double Word, vier Bytes zu übermitteltem Parameterwert zusammenfassen
           #pwWordHigh := SHL(IN := BYTE_TO_WORD(#sxRespParaMulti.sxData[3]), N := 8);
           #pwWordLow := BYTE_TO_WORD(#sxRespParaMulti.sxData[4]);
           #pwWord1 := #pwWordHigh XOR #pwWordLow;

           #pwWordHigh := SHL(IN := BYTE_TO_WORD(#sxRespParaMulti.sxData[5]), N := 8);
           #pwWordLow := BYTE_TO_WORD(#sxRespParaMulti.sxData[6]);
           #pwWord2 := #pwWordHigh XOR #pwWordLow;

           #pdDWordHigh := SHL(IN := WORD_TO_DWORD(#pwWord1), N := 16);
           #pdDWordLow := WORD_TO_DWORD(#pwWord2);

           // ermittelter Parameterwert eintragen (Word)
           #ValueRead1 := 0.0;
           #ValueRead2 := DWORD_TO_DINT(#pdDWordHigh XOR #pdDWordLow);

           // ermittelte Fehlernummer im Puffer zurücksetzen
           #ErrorNo := W#16#00;

           // Die Fehlerhaftigkeit des erkannten Parameter in der Fehlernummer löschen   
           #swParaError := #swParaError AND W#16#FFFE;

           // Format = Double Word ? = > gesendeter Parameter vier Bytes lang (FloatingPoint)
         ELSIF (#sxRespParaMulti.sxData[1] = B#16#08) THEN

           // Format = Double Word, vier Bytes zu übermitteltem Parameterwert zusammenfassen
           #pwWordHigh := SHL(IN := BYTE_TO_WORD(#sxRespParaMulti.sxData[3]), N := 8);
           #pwWordLow := BYTE_TO_WORD(#sxRespParaMulti.sxData[4]);
           #pwWord1 := #pwWordHigh XOR #pwWordLow;

           #pwWordHigh := SHL(IN := BYTE_TO_WORD(#sxRespParaMulti.sxData[5]), N := 8);
           #pwWordLow := BYTE_TO_WORD(#sxRespParaMulti.sxData[6]);
           #pwWord2 := #pwWordHigh XOR #pwWordLow;

           #pdDWordHigh := SHL(IN := WORD_TO_DWORD(#pwWord1), N := 16);
           #pdDWordLow := WORD_TO_DWORD(#pwWord2);

           // ermittelter Parameterwert eintragen (Word)
           #ValueRead1 := DWORD_TO_REAL(#pdDWordHigh XOR #pdDWordLow);
           #ValueRead2 := 0;

           // ermittelte Fehlernummer im Puffer zurücksetzen
           #ErrorNo := W#16#00;

           // Die Fehlerhaftigkeit des erkannten Parameter in der Fehlernummer löschen   
           #swParaError := #swParaError AND W#16#FFFE;

           // Unbekanter Datentyp
         ELSE

           #siErrorId := 5;
           #sbError := True;
           #sbDone := False;
           // Die Fehlerhaftigkeit des erkannten Parameter in der Fehlernummer eintragen   
           #swParaError := #swParaError OR W#16#01;

         END_IF;

         // Fehlerkennung zurücknehmen
         IF (#siErrorId = 3) OR (#siErrorId = 1) THEN
           #siErrorId := 0;
           #sbError := False;
         END_IF;

         #DiagId := W#16#00;

         // Auftrag : Parameter lesen ist abgeschlossen
         #sbRdStart := False;
         #sbRead := False;
       END_IF; // kein Fehler beim LESEN AZYKLISCH und Auftrag fertig 
     END_IF; // vom Auftrag "Parameter lesen" die Antwort abwarten und dann auswerten 
   END_IF; // Auftrag "Parameter lesen" wurde ausgelöst

   // Auftrag "Parameter schreiben" wurde ausgelöst
   IF #sbParaNo AND NOT #sbRead AND #sbWrite THEN

     // Auftrag "Parameter schreiben" bzw. "ändern" besteht aus zwei Aufträgen
     // 1. Teilauftrag "Parameter lesen"
     // 2. Teilauftrag "Parameter schreiben bzw. ändern"

     // 1. Teilauftrag "Parameter lesen" vorbereiten und abschicken
     IF #sbWrStart1 THEN

       // Ablöschen des Sendepuffers
       // Parameternummer des Parameters 
       #sxReqParaMulti.sxParaAdress.siParaNo := 0;

       // Subindex des Parameters
       #sxReqParaMulti.sxParaAdress.siIndex := 0;

       // Auftrags-HEADER erstellen
       // Auftragsreferenz
       #sxReqParaMulti.sxHeader.syReqRef := INT_TO_BYTE(#siReqRef);

       // Auftragskennung 0x01=Request Parameters
       #sxReqParaMulti.sxHeader.syReqId := B#16#01;

       // Achse
       #sxReqParaMulti.sxHeader.syAxisNo := #syAxisNo;

       // Anzahl Parameter        
       #sxReqParaMulti.sxHeader.syParaNo := B#16#01;

       // Auftrags-PARAMETERADRESSE erstellen
       // Parameternummer des Parameters                                
       #sxReqParaMulti.sxParaAdress.siParaNo := #Parameter;

       // Subindex des Parameters
       #sxReqParaMulti.sxParaAdress.siIndex := #Index;

       // SCHREIBEN AZYKLISCH
       #piLenTele := #siLenHeader + #siLenParaMulti;
       #WRREC_1(REQ := True,                                // Startimpuls
                ID := #hardwareId,                         // Diagnoseadresse
                INDEX := 47,                                  // Rahmentyp
                LEN := INT_TO_UINT(#piLenTele),             // maximale Länge
                DONE => #sbWrDone,                           // Schreibauftrag beendet
                BUSY => #sbWrBusy,                           // Slave beschäftigt
                ERROR => #sbWrError,                          // Fehler beim Schreiben
                STATUS => #pdStatus,                           // Status[1] = Error => Status[2] Error Decode + Status[3] Error Code
                RECORD := #sxReqParaMulti);                    // Zeiger auf zu schreibenen Datensatz

       // Ausgänge setzen
       #sbBusy := #sbWrBusy;
       #sbDone := #sbWrDone;

       // Fehler auswerten
       IF #sbWrError THEN

         // Fehlerstatus aus dem Doppelwort filtern und weitergeben                
         #pwWord1 := DWORD_TO_WORD(SHR(IN := (#pdStatus AND DW#16#FFFF00), N := 8));

         // Fehlerstatus setzen
         #siErrorId := 3;
         #DiagId := #pwWord1;

         //Temporärer Fehler: #pdStatus = 80A7, 80B5, 80C0, 80C1, 80C2, 80C3 oder 80C4 zulassen und nocheinmal versuchen
         IF NOT (#pwWord1 = DW#16#80A7) AND NOT (#pwWord1 = DW#16#80B5) AND NOT (#pwWord1 = DW#16#80C0) AND
           NOT (#pwWord1 = DW#16#80C1) AND NOT (#pwWord1 = DW#16#80C2) AND NOT (#pwWord1 = DW#16#80C3) AND
           NOT (#pwWord1 = DW#16#80C4) THEN

           // Wiederholungsauftrag wieder zurücknehmen
           #sbWrStart1 := False;
           #sbRdStart1 := False;
           #sbWrite := False;

           // Fehler ausgeben 
           #sbError := #sbWrError;

         ELSE
           // Fehlerwiederholauftrag ??                   
           IF #siErrorCount = #siMaxErrCount THEN

             // Wiederholungsauftrag wieder zurücknehmen
             #sbWrStart1 := False;
             #sbRdStart1 := False;
             #sbWrite := False;

             //Fehlerzähler zurücksetzen
             #siErrorCount := 0;


             // Fehler ausgeben 
             #sbError := #sbWrError;
             // nix tun bis Zähler überläuft
           ELSE
             #siErrorCount := #siErrorCount + 1;
           END_IF;
         END_IF;

         // kein Fehler beim SCHEIBEN AZYKLISCH und Auftrag fertig 
       ELSIF NOT #sbWrBusy AND #sbWrDone THEN

         // Fehlerkennung zurücknehmen
         IF (#siErrorId = 3) THEN
           #siErrorId := 0;
           #sbError := False;
         END_IF;

         #DiagId := W#16#00;

         // Schreibauftrag fertig melden und Leseantrag anstossen
         #sbWrStart1 := False;
         #sbRdStart1 := True;
       END_IF;
     END_IF; // 1. Teilauftrag "Parameter lesen" vorbereiten und abschicken

     // vom 1. Teilauftrag "Parameter lesen" die Antwort abwarten und dann auswerten
     IF #sbRdStart1 THEN

       // Ablöschen des Empfangspuffers
       #sxRespParaMulti.sxHeader.syReqRef := B#16#00;
       #sxRespParaMulti.sxHeader.syReqId := B#16#00;
       #sxRespParaMulti.sxHeader.syAxisNo := B#16#00;
       #sxRespParaMulti.sxHeader.syParaNo := B#16#00;

       FOR #piCount := 1 TO #siLenParaMulti DO
         #sxRespParaMulti.sxData[#piCount] := B#16#00;
       END_FOR;

       // LESEN AZYKLISCH
       #piLenTele := #siLenHeader + #siLenParaMulti;
       #RDREC_1(REQ := True,                                // Startimpuls
                ID := #hardwareId,                         // Diagnoseadresse        
                INDEX := 47,                                  // Rahmentyp           
                MLEN := INT_TO_UINT(#piLenTele),             // maximale Länge
                VALID => #pbValidSFB,                         // neuer Datensatz empfangen und gültig      
                BUSY => #sbRdBusy,                           // Slave beschäftigt
                ERROR => #sbRdError,                          // Fehler beim Schreiben
                STATUS => #pdStatus,                           // Status[1] = Error => Status[2] Error Decode + Status[3] Error Code 
                LEN => #piLenSFB,                           // Länge des gelesenen Datensatzes
                RECORD := #sxRespParaMulti);                   // Zeiger auf gelesenen Datensatz

       // Ausgänge setzen
       #sbBusy := #sbRdBusy;
       #sbDone := #pbValidSFB;

       // Fehler auswerten
       IF #sbRdError THEN
         // Fehlerstatus aus dem Doppelwort filtern und weitergeben                
         #pwWord1 := DWORD_TO_WORD(SHR(IN := (#pdStatus AND DW#16#FFFF00), N := 8));

         // Fehlerstatus setzen
         #siErrorId := 3;
         #DiagId := #pwWord1;

         //Temporärer Fehler: #pdStatus = 80A7, 80B5, 80C0, 80C1, 80C2, 80C3 oder 80C4 zulassen und nocheinmal versuchen
         IF NOT (#pwWord1 = DW#16#80A7) AND NOT (#pwWord1 = DW#16#80B5) AND NOT (#pwWord1 = DW#16#80C0) AND
           NOT (#pwWord1 = DW#16#80C1) AND NOT (#pwWord1 = DW#16#80C2) AND NOT (#pwWord1 = DW#16#80C3) AND
           NOT (#pwWord1 = DW#16#80C4) THEN

           // Wiederholungsauftrag wieder zurücknehmen
           #sbWrStart1 := False;
           #sbRdStart1 := False;
           #sbWrite := False;

           // Fehler ausgeben 
           #sbError := #sbRdError;

         ELSE
           // Fehlerwiederholauftrag ??                   
           IF #siErrorCount = #siMaxErrCount THEN

             // Wiederholungsauftrag wieder zurücknehmen
             #sbWrStart1 := False;
             #sbRdStart1 := False;
             #sbWrite := False;

             //Fehlerzähler zurücksetzen
             #siErrorCount := 0;


             // Fehler ausgeben 
             #sbError := #sbRdError;

             // nix tun bis Zähler überläuft
           ELSE
             #siErrorCount := #siErrorCount + 1;
           END_IF;
         END_IF;

         // Fehler : die Auftragsreferenz der Antwort übertimmt nicht mit der Auftragsreferenz der Anfrage überein
       ELSIF NOT (#siReqRef = BYTE_TO_INT(#sxRespParaMulti.sxHeader.syReqRef)) AND NOT #sbRdBusy AND #pbValidSFB THEN
         #siErrorId := 1;
         #sbError := True;
         #sbDone := False;

         // Wiederholungsauftrag wieder zurücknehmen
         #sbWrStart1 := False;
         #sbRdStart1 := False;
         #sbWrite := False;

         // Fehler : falsche Auftragskennung zurück erhalten    
       ELSIF NOT (#sxRespParaMulti.sxHeader.syReqId = B#16#81 OR #sxRespParaMulti.sxHeader.syReqId = B#16#01) AND
         NOT #sbRdBusy AND #pbValidSFB THEN
         #siErrorId := 1;
         #sbError := True;
         #sbDone := False;

         // Wiederholungsauftrag wieder zurücknehmen
         #sbWrStart1 := False;
         #sbRdStart1 := False;
         #sbWrite := False;

         // Fehler : die angeforderte Anzahl Parameter entspricht nicht der übermittelten Anzahl Parameter überein
       ELSIF NOT (#sxRespParaMulti.sxHeader.syParaNo = B#16#01) AND NOT #sbRdBusy AND #pbValidSFB THEN
         #siErrorId := 1;
         #sbError := True;
         #sbDone := False;

         // Wiederholungsauftrag wieder zurücknehmen
         #sbWrStart1 := False;
         #sbRdStart1 := False;
         #sbWrite := False;

         // Fehler : die Achse entspricht nicht der übergebenen Achse
       ELSIF NOT (#syAxisNo = #sxRespParaMulti.sxHeader.syAxisNo) AND NOT #sbRdBusy AND #pbValidSFB THEN
         #siErrorId := 1;
         #sbError := True;
         #sbDone := False;

         // Wiederholungsauftrag wieder zurücknehmen
         #sbWrStart1 := False;
         #sbRdStart1 := False;
         #sbWrite := False;

         // kein Fehler beim LESEN AZYKLISCH und Auftrag fertig 
       ELSIF NOT #sbRdBusy AND #pbValidSFB THEN

         // die angefragten Parameter auswerten und im Puffer abspeichern
         // ermitteltes Format des Parameters abspeichern
         #syFormat := #sxRespParaMulti.sxData[1];

         // Format = Error ? = > gesendeter Parameter fehlerhaft
         IF (BYTE_TO_INT(#sxRespParaMulti.sxData[1]) = 68) THEN

           // Format = Error, zwei Bytes zu übermittelten Fehlernummer zusammenfassen
           #pwWordHigh := SHL(IN := BYTE_TO_WORD(#sxRespParaMulti.sxData[3]), N := 8);
           #pwWordLow := BYTE_TO_WORD(#sxRespParaMulti.sxData[4]);

           #sbError := True;

           // ermittelte Fehlernummer im Puffer abspeichern
           #ErrorNo := #pwWordHigh XOR #pwWordLow;

           // Die Fehlerhaftigkeit des erkannten Parameter in der Fehlernummer eintragen   
           #swParaError := #swParaError OR W#16#01;

           // Format = Byte ? = > gesendeter Parameter ein Byte lang
         ELSIF (#sxRespParaMulti.sxData[1] = B#16#41) OR
           (#sxRespParaMulti.sxData[1] = B#16#02) OR (#sxRespParaMulti.sxData[1] = B#16#05) THEN

           // ermittelte Fehlernummer im Puffer zurücksetzen
           #ErrorNo := W#16#00;

           // Die Fehlerhaftigkeit des erkannten Parameter in der Fehlernummer löschen   
           #swParaError := #swParaError AND W#16#FFFE;

           // Format = Word ? = > gesendeter Parameter zwei Bytes lang
         ELSIF (#sxRespParaMulti.sxData[1] = B#16#42) OR (#sxRespParaMulti.sxData[1] = B#16#03)
           OR (#sxRespParaMulti.sxData[1] = B#16#06) OR (#sxRespParaMulti.sxData[1] = B#16#0A) THEN

           // ermittelte Fehlernummer im Puffer zurücksetzen
           #ErrorNo := W#16#00;

           // Die Fehlerhaftigkeit des erkannten Parameter in der Fehlernummer löschen   
           #swParaError := #swParaError AND W#16#FFFE;


           // Format = Double Word ? = > gesendeter Parameter vier Bytes lang
         ELSIF (#sxRespParaMulti.sxData[1] = B#16#43) OR (#sxRespParaMulti.sxData[1] = B#16#04) OR
           (#sxRespParaMulti.sxData[1] = B#16#07) OR (#sxRespParaMulti.sxData[1] = B#16#08) OR
           (#sxRespParaMulti.sxData[1] = B#16#0D) THEN

           // ermittelte Fehlernummer im Puffer zurücksetzen
           #ErrorNo := W#16#00;

           // Die Fehlerhaftigkeit des erkannten Parameter in der Fehlernummer löschen   
           #swParaError := #swParaError AND W#16#FFFE;

           // Unbekanter Datentyp
         ELSE

           #siErrorId := 5;
           #sbError := True;
           #sbDone := False;
           // Die Fehlerhaftigkeit des erkannten Parameter in der Fehlernummer eintragen   
           #swParaError := #swParaError OR W#16#01;

         END_IF;

         // Fehlerkennung zurücknehmen
         IF (#siErrorId = 3) OR (#siErrorId = 1) THEN
           #siErrorId := 0;
           #sbError := False;
         END_IF;

         #DiagId := W#16#00;

         // 1. Teilauftrag "Parameter lesen" ist abgeschlossen
         #sbRdStart1 := False;

         // einer der gesendeten Parameter ist fehlerhaft => Abbruch, kein "Parameter schreiben" erforderlich
         IF (#swParaError = W#16#00) THEN
           #sbWrStart2 := True;
         ELSE
           #sbWrStart2 := False;
         END_IF;
       END_IF; // kein Fehler beim LESEN AZYKLISCH und Auftrag fertig 
     END_IF; // vom 1. Teilauftrag "Parameter lesen" die Antwort abwarten und dann auswerten 

     // 2. Teilauftrag "Parameter schreiben bzw. ändern" vorbereiten und abschicken
     IF #sbWrStart2 THEN

       // Ablöschen des Sendepuffers            
       FOR #piCount := 1 TO #siLenChaPara DO
         // Parameteradresse und Parameterwert des Parameters 
         #sxChaParaMulti.sxData[#piCount] := B#16#00;
       END_FOR;

       // Auftrags-HEADER erstellen
       // Auftragsreferenz
       #sxChaParaMulti.sxHeader.syReqRef := INT_TO_BYTE(#siReqRef);

       // Auftragskennung 0x01=Request Parameters | 0x02=Change Parameters
       #sxChaParaMulti.sxHeader.syReqId := B#16#02;

       // Achse
       #sxChaParaMulti.sxHeader.syAxisNo := #syAxisNo;

       // Anzahl Parameter        
       #sxChaParaMulti.sxHeader.syParaNo := B#16#01;

       // Auftrags-PARAMETERADRESSE erstellen                
       // Attribute of parameters (0x10=Value, 0x30=Text)
       #sxChaParaMulti.sxData[1] := B#16#10;

       // No. of elements (DEC: for single elements=1) 
       #sxChaParaMulti.sxData[2] := B#16#01;

       // Parameternummer des Parameters                                
       #sxChaParaMulti.sxData[4] := INT_TO_BYTE(#Parameter);
       #sxChaParaMulti.sxData[3] := WORD_TO_BYTE(SHR(IN := INT_TO_WORD(#Parameter), N := 8));

       // Subindex des Parameters
       #sxChaParaMulti.sxData[6] := INT_TO_BYTE(#Index);
       #sxChaParaMulti.sxData[5] := WORD_TO_BYTE(SHR(IN := INT_TO_WORD(#Index), N := 8));

       // Auftrags-PARAMETERVALUE erstellen    
       // Format (BYTE, WORD, DWORD des Parameterwert übergeben
       #sxChaParaMulti.sxData[7] := #syFormat;

       // Number of value
       #sxChaParaMulti.sxData[8] := B#16#01;

       // Value of parameter in Bytes
       IF (#syFormat = B#16#41) OR
         (#syFormat = B#16#02) OR (#syFormat = B#16#05) THEN

         #sxChaParaMulti.sxData[9] := WORD_TO_BYTE(DWORD_TO_WORD(DINT_TO_DWORD(REAL_TO_DINT(#ValueWrite1))));
         #sxChaParaMulti.sxData[10] := 16#00;  //WORD_TO_BYTE(DWORD_TO_WORD(SHR(IN := DINT_TO_DWORD(REAL_TO_DINT(#ValueWrite1)), N := 8)));

         // Value of parameter in Word
       ELSIF (#syFormat = B#16#42) OR (#syFormat = B#16#03) OR
         (#syFormat = B#16#06) OR (#syFormat = B#16#0A) THEN

         #sxChaParaMulti.sxData[10] := WORD_TO_BYTE(DWORD_TO_WORD(DINT_TO_DWORD(REAL_TO_DINT(#ValueWrite1))));
         #sxChaParaMulti.sxData[9] := WORD_TO_BYTE(DWORD_TO_WORD(SHR(IN := DINT_TO_DWORD(REAL_TO_DINT(#ValueWrite1)), N := 8)));

         // Value of parameter in DWord    
       ELSIF (#syFormat = B#16#43) OR (#syFormat = B#16#04) OR
         (#syFormat = B#16#07) OR (#syFormat = B#16#0D) THEN

         #sxChaParaMulti.sxData[12] := WORD_TO_BYTE(DWORD_TO_WORD(DINT_TO_DWORD(#ValueWrite2)));
         #sxChaParaMulti.sxData[11] := WORD_TO_BYTE(DWORD_TO_WORD(SHR(IN := DINT_TO_DWORD(#ValueWrite2), N := 8)));
         #sxChaParaMulti.sxData[10] := WORD_TO_BYTE(DWORD_TO_WORD(SHR(IN := DINT_TO_DWORD(#ValueWrite2), N := 16)));
         #sxChaParaMulti.sxData[9] := WORD_TO_BYTE(DWORD_TO_WORD(SHR(IN := DINT_TO_DWORD(#ValueWrite2), N := 24)));


         // Value of parameter in DWord (FloatingPoint)   
       ELSIF (#syFormat = B#16#08) THEN

         #sxChaParaMulti.sxData[12] := WORD_TO_BYTE(DWORD_TO_WORD(REAL_TO_DWORD(#ValueWrite1)));
         #sxChaParaMulti.sxData[11] := WORD_TO_BYTE(DWORD_TO_WORD(SHR(IN := REAL_TO_DWORD(#ValueWrite1), N := 8)));
         #sxChaParaMulti.sxData[10] := WORD_TO_BYTE(DWORD_TO_WORD(SHR(IN := REAL_TO_DWORD(#ValueWrite1), N := 16)));
         #sxChaParaMulti.sxData[9] := WORD_TO_BYTE(DWORD_TO_WORD(SHR(IN := REAL_TO_DWORD(#ValueWrite1), N := 24)));

       END_IF;

       // SCHREIBEN AZYKLISCH
       #piLenTele := #siLenHeader + #siLenChaPara;
       #WRREC_1(REQ := True,                                // Startimpuls
                ID := #hardwareId,                         // Diagnoseadresse
                INDEX := 47,                                  // Rahmentyp
                LEN := INT_TO_UINT(#piLenTele),             // maximale Länge
                DONE => #sbWrDone,                           // Schreibauftrag beendet
                BUSY => #sbWrBusy,                           // Slave beschäftigt
                ERROR => #sbWrError,                          // Fehler beim Schreiben
                STATUS => #pdStatus,                           // Status[1] = Error => Status[2] Error Decode + Status[3] Error Code
                RECORD := #sxChaParaMulti);                    // Zeiger auf zu schreibenen Datensatzes

       // Ausgänge setzen
       #sbBusy := #sbWrBusy;
       #sbDone := #sbWrDone;

       // Fehler auswerten
       IF #sbWrError THEN
         // Fehlerstatus aus dem Doppelwort filtern und weitergeben                
         #pwWord1 := DWORD_TO_WORD(SHR(IN := (#pdStatus AND DW#16#FFFF00), N := 8));

         // Fehlerstatus setzen
         #siErrorId := 3;
         #sbError := False;
         #DiagId := #pwWord1;

         //Temporärer Fehler: #pdStatus = 80A7, 80B5, 80C0, 80C1, 80C2, 80C3 oder 80C4 zulassen und nocheinmal versuchen
         IF NOT (#pwWord1 = DW#16#80A7) AND NOT (#pwWord1 = DW#16#80B5) AND NOT (#pwWord1 = DW#16#80C0) AND
           NOT (#pwWord1 = DW#16#80C1) AND NOT (#pwWord1 = DW#16#80C2) AND NOT (#pwWord1 = DW#16#80C3) AND
           NOT (#pwWord1 = DW#16#80C4) THEN

           // Wiederholungsauftrag wieder zurücknehmen
           #sbWrStart2 := False;
           #sbRdStart2 := False;
           #sbWrite := False;

           // Fehler ausgeben 
           #sbError := #sbWrError;

         ELSE
           // Fehlerwiederholauftrag ??                   
           IF #siErrorCount = #siMaxErrCount THEN

             // Wiederholungsauftrag wieder zurücknehmen
             #sbWrStart2 := False;
             #sbRdStart2 := False;
             #sbWrite := False;

             //Fehlerzähler zurücksetzen
             #siErrorCount := 0;


             // Fehler ausgeben 
             #sbError := #sbWrError;

             // nix tun bis Zähler überläuft
           ELSE
             #siErrorCount := #siErrorCount + 1;
           END_IF;
         END_IF;

         // kein Fehler beim SCHEIBEN AZYKLISCH und Auftrag fertig 
       ELSIF NOT #sbWrBusy AND #sbWrDone THEN
         // Fehlerkennung zurücknehmen
         #DiagId := W#16#00;

         // Schreibauftrag fertig melden und Leseantrag anstossen
         #sbWrStart2 := False;
         #sbRdStart2 := True;
       END_IF;
     END_IF; // 2. Teilauftrag "Parameter schreiben bzw. ändern" vorbereiten und abschicken

     // vom 2. Teilauftrag "Parameter schreiben bzw. ändern" die Antwort abwarten und dann auswerten
     IF #sbRdStart2 THEN

       // Ablöschen des Empfangspuffers
       #sxRespParaMulti.sxHeader.syReqRef := B#16#00;
       #sxRespParaMulti.sxHeader.syReqId := B#16#00;
       #sxRespParaMulti.sxHeader.syAxisNo := B#16#00;
       #sxRespParaMulti.sxHeader.syParaNo := B#16#00;

       FOR #piCount := 1 TO #siLenParaMulti DO
         #sxRespParaMulti.sxData[#piCount] := B#16#00;
       END_FOR;

       // LESEN AZYKLISCH
       #piLenTele := #siLenHeader + #siLenParaMulti;
       #RDREC_1(REQ := True,                                // Startimpuls
                ID := #hardwareId,                         // Diagnoseadresse        
                INDEX := 47,                                  // Rahmentyp           
                MLEN := INT_TO_UINT(#piLenTele),             // maximale Länge
                VALID => #pbValidSFB,                         // neuer Datensatz empfangen und gültig   
                BUSY => #sbRdBusy,                           // Slave beschäftigt
                ERROR => #sbRdError,                          // Fehler beim Schreiben
                STATUS => #pdStatus,                           // Status[1] = Error => Status[2] Error Decode + Status[3] Error Code 
                LEN => #piLenSFB,                           // Länge des gelesenen Datensatzes
                RECORD := #sxRespParaMulti);                   // Zeiger auf gelesenen Datensatz

       // Ausgänge setzen
       #sbBusy := #sbRdBusy;
       #sbDone := #pbValidSFB;

       // Fehler auswerten
       IF #sbRdError THEN
         // Fehlerstatus aus dem Doppelwort filtern und weitergeben                
         #pwWord1 := DWORD_TO_WORD(SHR(IN := (#pdStatus AND DW#16#FFFF00), N := 8));

         // Fehlerstatus setzen
         #siErrorId := 3;
         #DiagId := #pwWord1;

